LIN {X 0,Y 105.055,Z 539.774,A -85,B 0,C 180,E1 -26170.459,E2 -26170.459} C_VEL
LIN {X 0,Y 104.648,Z 537.475,A -85,B 0,C 180,E1 -26178.377,E2 -26178.377} C_VEL
LIN {X 0,Y 105.683,Z 533.747,A -85,B 0,C 180,E1 -26186.188,E2 -26186.188} C_VEL
LIN {X 0,Y 107.046,Z 529.972,A -85,B 0,C 180,E1 -26191.882,E2 -26191.882} C_VEL
LIN {X 0,Y 109.151,Z 525.302,A -85,B 0,C 180,E1 -26197.399,E2 -26197.399} C_VEL
LIN {X 0,Y 112.696,Z 518.5,A -85,B 0,C 180,E1 -26203.525,E2 -26203.525} C_VEL
LIN {X 0,Y 116.604,Z 511.397,A -85,B 0,C 180,E1 -26208.447,E2 -26208.447} C_VEL
LIN {X 0,Y 121.232,Z 502.855,A -85,B 0,C 180,E1 -26213.036,E2 -26213.036} C_VEL
LIN {X 0,Y 126.13,Z 493.405,A -85,B 0,C 180,E1 -26216.946,E2 -26216.946} C_VEL
LIN {X 0,Y 130.9,Z 483.256,A -85,B 0,C 180,E1 -26220.221,E2 -26220.221} C_VEL
LIN {X 0,Y 135.895,Z 470.856,A -85,B 0,C 180,E1 -26223.331,E2 -26223.331} C_VEL
LIN {X 0,Y 139.577,Z 460.327,A -85,B 0,C 180,E1 -26225.383,E2 -26225.383} C_VEL
LIN {X 0,Y 143.441,Z 448.136,A -85,B 0,C 180,E1 -26227.103,E2 -26227.103} C_VEL
LIN {X 0,Y 146.585,Z 434.369,A -85,B 0,C 180,E1 -26228.641,E2 -26228.641} C_VEL
LIN {X 0,Y 148.972,Z 420.343,A -85,B 0,C 180,E1 -26229.683,E2 -26229.683} C_VEL
LIN {X 0,Y 150.699,Z 403.652,A -85,B 0,C 180,E1 -26230.423,E2 -26230.423} C_VEL
LIN {X 0,Y 154.161,Z 361.132,A -85,B 0,C 180,E1 -26231.967,E2 -26231.967} C_VEL
LIN {X 0,Y 149.223,Z 350.379,A -85,B 0,C 180,E1 -26235.125,E2 -26235.125} C_VEL
LIN {X 0,Y 143.968,Z 340.636,A -85,B 0,C 180,E1 -26238.855,E2 -26238.855} C_VEL
LIN {X 0,Y 139.833,Z 333.875,A -85,B 0,C 180,E1 -26242.202,E2 -26242.202} C_VEL
LIN {X 0,Y 137.16,Z 329.846,A -85,B 0,C 180,E1 -26244.64,E2 -26244.64} C_VEL
LIN {X 0,Y 135.135,Z 326.776,A -85,B 0,C 180,E1 -26246.702,E2 -26246.702} C_VEL
LIN {X 0,Y 132.21,Z 322.641,A -85,B 0,C 180,E1 -26250.064,E2 -26250.064} C_VEL
LIN {X 0,Y 129.671,Z 319.416,A -85,B 0,C 180,E1 -26253.506,E2 -26253.506} C_VEL
LIN {X 0,Y 128.977,Z 318.09,A -85,B 0,C 180,E1 -26254.659,E2 -26254.659} C_VEL
LIN {X 0,Y 126.508,Z 315.752,A -85,B 0,C 180,E1 -26259.081,E2 -26259.081} C_VEL
LIN {X 0,Y 125.34,Z 312.869,A -85,B 0,C 180,E1 -26262.402,E2 -26262.402} C_VEL
LIN {X 0,Y 123.472,Z 311.706,A -85,B 0,C 180,E1 -26273.468,E2 -26273.468} C_VEL
LIN {X 0,Y 124.564,Z 312.157,A -85,B 0,C 180,E1 -26280.716,E2 -26280.716} C_VEL
LIN {X 0,Y 125.644,Z 313.032,A -85,B 0,C 180,E1 -26284.014,E2 -26284.014} C_VEL
LIN {X 0,Y 127.576,Z 316.671,A -85,B 0,C 180,E1 -26288.599,E2 -26288.599} C_VEL
LIN {X 0,Y 129.318,Z 318.362,A -85,B 0,C 180,E1 -26291.474,E2 -26291.474} C_VEL
LIN {X 0,Y 131.665,Z 322.03,A -85,B 0,C 180,E1 -26294.889,E2 -26294.889} C_VEL
LIN {X 0,Y 132.836,Z 323.455,A -85,B 0,C 180,E1 -26296.328,E2 -26296.328} C_VEL
LIN {X 0,Y 136.355,Z 328.602,A -85,B 0,C 180,E1 -26300.191,E2 -26300.191} C_VEL
LIN {X 0,Y 139.525,Z 333.327,A -85,B 0,C 180,E1 -26303.148,E2 -26303.148} C_VEL
LIN {X 0,Y 144.459,Z 341.575,A -85,B 0,C 180,E1 -26307.146,E2 -26307.146} C_VEL
LIN {X 0,Y 147.72,Z 347.787,A -85,B 0,C 180,E1 -26309.508,E2 -26309.508} C_VEL
LIN {X 0,Y 152.037,Z 359.604,A -85,B 0,C 180,E1 -26312.582,E2 -26312.582} C_VEL
LIN {X 0,Y 153.923,Z 365.668,A -85,B 0,C 180,E1 -26313.879,E2 -26313.879} C_VEL
LIN {X 0,Y 149.419,Z 421.282,A -85,B 0,C 180,E1 -26316.014,E2 -26316.014} C_VEL
LIN {X 0,Y 147.033,Z 436.247,A -85,B 0,C 180,E1 -26316.953,E2 -26316.953} C_VEL
LIN {X 0,Y 144.373,Z 447.938,A -85,B 0,C 180,E1 -26318.002,E2 -26318.002} C_VEL
LIN {X 0,Y 140.529,Z 461.489,A -85,B 0,C 180,E1 -26319.744,E2 -26319.744} C_VEL
LIN {X 0,Y 136.243,Z 473.608,A -85,B 0,C 180,E1 -26321.808,E2 -26321.808} C_VEL
LIN {X 0,Y 131.776,Z 485.158,A -85,B 0,C 180,E1 -26324.504,E2 -26324.504} C_VEL
LIN {X 0,Y 127.567,Z 494.106,A -85,B 0,C 180,E1 -26327.018,E2 -26327.018} C_VEL
LIN {X 0,Y 122.362,Z 504.452,A -85,B 0,C 180,E1 -26330.818,E2 -26330.818} C_VEL
LIN {X 0,Y 117.437,Z 513.807,A -85,B 0,C 180,E1 -26335.353,E2 -26335.353} C_VEL
LIN {X 0,Y 113.067,Z 521.924,A -85,B 0,C 180,E1 -26340.491,E2 -26340.491} C_VEL
LIN {X 0,Y 109.983,Z 528.046,A -85,B 0,C 180,E1 -26345.458,E2 -26345.458} C_VEL
LIN {X 0,Y 107.481,Z 533.33,A -85,B 0,C 180,E1 -26350.917,E2 -26350.917} C_VEL
LIN {X 0,Y 105.951,Z 537.632,A -85,B 0,C 180,E1 -26356.575,E2 -26356.575} C_VEL
LIN {X 0,Y 105.213,Z 541.041,A -85,B 0,C 180,E1 -26362.322,E2 -26362.322} C_VEL
LIN {X 0,Y 105.226,Z 544.198,A -85,B 0,C 180,E1 -26370,E2 -26370} C_VEL
LIN {X 0,Y 105.107,Z 545.222,A -85,B 0,C 180,E1 -26373.833,E2 -26373.833} C_VEL
LIN {X 0,Y 105.686,Z 546.264,A -85,B 0,C 180,E1 -26381.507,E2 -26381.507} C_VEL
LIN {X 0,Y 107.772,Z 546.007,A -85,B 0,C 180,E1 -26389.029,E2 -26389.029} C_VEL
LIN {X 0,Y 111.648,Z 544.464,A -85,B 0,C 180,E1 -26396.143,E2 -26396.143} C_VEL
LIN {X 0,Y 117.254,Z 541.466,A -85,B 0,C 180,E1 -26402.944,E2 -26402.944} C_VEL
LIN {X 0,Y 122.733,Z 538.083,A -85,B 0,C 180,E1 -26407.779,E2 -26407.779} C_VEL
LIN {X 0,Y 125.139,Z 536.162,A -85,B 0,C 180,E1 -26410.108,E2 -26410.108} C_VEL
LIN {X 0,Y 127.914,Z 532.718,A -85,B 0,C 180,E1 -26414.149,E2 -26414.149} C_VEL
LIN {X 0,Y 131.209,Z 528.811,A -85,B 0,C 180,E1 -26417.901,E2 -26417.901} C_VEL
LIN {X 0,Y 134.288,Z 526.052,A -85,B 0,C 180,E1 -26419.712,E2 -26419.712} C_VEL
LIN {X 0,Y 142.813,Z 518.685,A -85,B 0,C 180,E1 -26423.097,E2 -26423.097} C_VEL
LIN {X 0,Y 152.062,Z 509.256,A -85,B 0,C 180,E1 -26426.294,E2 -26426.294} C_VEL
LIN {X 0,Y 158.977,Z 501.172,A -85,B 0,C 180,E1 -26428.318,E2 -26428.318} C_VEL
LIN {X 0,Y 166.918,Z 490.585,A -85,B 0,C 180,E1 -26430.271,E2 -26430.271} C_VEL
LIN {X 0,Y 174.225,Z 478.929,A -85,B 0,C 180,E1 -26431.931,E2 -26431.931} C_VEL
LIN {X 0,Y 180.261,Z 467.528,A -85,B 0,C 180,E1 -26433.103,E2 -26433.103} C_VEL
LIN {X 0,Y 185.569,Z 455.21,A -85,B 0,C 180,E1 -26434.086,E2 -26434.086} C_VEL
LIN {X 0,Y 189.847,Z 442.69,A -85,B 0,C 180,E1 -26434.817,E2 -26434.817} C_VEL
LIN {X 0,Y 193.446,Z 428.393,A -85,B 0,C 180,E1 -26435.413,E2 -26435.413} C_VEL
LIN {X 0,Y 195.769,Z 413.722,A -85,B 0,C 180,E1 -26435.832,E2 -26435.832} C_VEL
LIN {X 0,Y 196.762,Z 403.98,A -85,B 0,C 180,E1 -26436.095,E2 -26436.095} C_VEL
LIN {X 0,Y 194.512,Z 396.884,A -85,B 0,C 180,E1 -26439.321,E2 -26439.321} C_VEL
LIN {X 0,Y 192.732,Z 391.862,A -85,B 0,C 180,E1 -26442.537,E2 -26442.537} C_VEL
LIN {X 0,Y 192.084,Z 390.368,A -85,B 0,C 180,E1 -26443.929,E2 -26443.929} C_VEL
LIN {X 0,Y 190.654,Z 386.905,A -85,B 0,C 180,E1 -26448.3,E2 -26448.3} C_VEL
LIN {X 0,Y 190.006,Z 386.116,A -85,B 0,C 180,E1 -26453.626,E2 -26453.626} C_VEL
LIN {X 0,Y 190.784,Z 386.681,A -85,B 0,C 180,E1 -26458.463,E2 -26458.463} C_VEL
LIN {X 0,Y 192.443,Z 390.776,A -85,B 0,C 180,E1 -26463.203,E2 -26463.203} C_VEL
LIN {X 0,Y 194.198,Z 394.785,A -85,B 0,C 180,E1 -26466.421,E2 -26466.421} C_VEL
LIN {X 0,Y 196.692,Z 400.396,A -85,B 0,C 180,E1 -26469.834,E2 -26469.834} C_VEL
LIN {X 0,Y 197,Z 401.105,A -85,B 0,C 180,E1 -26470.207,E2 -26470.207} C_VEL
LIN {X 0,Y 194.942,Z 418.493,A -85,B 0,C 180,E1 -26470.687,E2 -26470.687} C_VEL
LIN {X 0,Y 192.039,Z 432.581,A -85,B 0,C 180,E1 -26471.22,E2 -26471.22} C_VEL
LIN {X 0,Y 187.985,Z 446.274,A -85,B 0,C 180,E1 -26471.97,E2 -26471.97} C_VEL
LIN {X 0,Y 183.008,Z 459.186,A -85,B 0,C 180,E1 -26472.982,E2 -26472.982} C_VEL
LIN {X 0,Y 177.404,Z 470.841,A -85,B 0,C 180,E1 -26474.182,E2 -26474.182} C_VEL
LIN {X 0,Y 170.672,Z 482.429,A -85,B 0,C 180,E1 -26475.737,E2 -26475.737} C_VEL
LIN {X 0,Y 162.454,Z 494.275,A -85,B 0,C 180,E1 -26477.875,E2 -26477.875} C_VEL
LIN {X 0,Y 155.149,Z 503.119,A -85,B 0,C 180,E1 -26479.963,E2 -26479.963} C_VEL
LIN {X 0,Y 147.053,Z 511.638,A -85,B 0,C 180,E1 -26482.617,E2 -26482.617} C_VEL
LIN {X 0,Y 138.654,Z 519.319,A -85,B 0,C 180,E1 -26485.885,E2 -26485.885} C_VEL
LIN {X 0,Y 129.874,Z 526.245,A -85,B 0,C 180,E1 -26490.026,E2 -26490.026} C_VEL
LIN {X 0,Y 122.973,Z 530.956,A -85,B 0,C 180,E1 -26494.039,E2 -26494.039} C_VEL
LIN {X 0,Y 116.733,Z 534.675,A -85,B 0,C 180,E1 -26498.496,E2 -26498.496} C_VEL
LIN {X 0,Y 109.621,Z 538.24,A -85,B 0,C 180,E1 -26505.154,E2 -26505.154} C_VEL
LIN {X 0,Y 104.048,Z 540.303,A -85,B 0,C 180,E1 -26512.563,E2 -26512.563} C_VEL
LIN {X 0,Y 100.166,Z 540.919,A -85,B 0,C 180,E1 -26520.586,E2 -26520.586} C_VEL
LIN {X 0,Y 98.12,Z 540.097,A -85,B 0,C 180,E1 -26529.015,E2 -26529.015} C_VEL
LIN {X 0,Y 97.645,Z 539.166,A -85,B 0,C 180,E1 -26533.269,E2 -26533.269} C_VEL
LIN {X 0,Y 97.801,Z 536.251,A -85,B 0,C 180,E1 -26541.737,E2 -26541.737} C_VEL
LIN {X 0,Y 98.952,Z 532.993,A -85,B 0,C 180,E1 -26548.208,E2 -26548.208} C_VEL
LIN {X 0,Y 101.292,Z 527.59,A -85,B 0,C 180,E1 -26555.974,E2 -26555.974} C_VEL
LIN {X 0,Y 104.589,Z 521.332,A -85,B 0,C 180,E1 -26562.615,E2 -26562.615} C_VEL
LIN {X 0,Y 109.112,Z 513.53,A -85,B 0,C 180,E1 -26568.787,E2 -26568.787} C_VEL
LIN {X 0,Y 113.87,Z 505.378,A -85,B 0,C 180,E1 -26573.652,E2 -26573.652} C_VEL
LIN {X 0,Y 119.328,Z 495.55,A -85,B 0,C 180,E1 -26578.11,E2 -26578.11} C_VEL
LIN {X 0,Y 124.289,Z 485.719,A -85,B 0,C 180,E1 -26581.537,E2 -26581.537} C_VEL
LIN {X 0,Y 129.531,Z 473.872,A -85,B 0,C 180,E1 -26584.729,E2 -26584.729} C_VEL
LIN {X 0,Y 133.264,Z 463.878,A -85,B 0,C 180,E1 -26586.861,E2 -26586.861} C_VEL
LIN {X 0,Y 137.612,Z 451.509,A -85,B 0,C 180,E1 -26588.727,E2 -26588.727} C_VEL
LIN {X 0,Y 141.054,Z 438.037,A -85,B 0,C 180,E1 -26590.37,E2 -26590.37} C_VEL
LIN {X 0,Y 143.774,Z 423.832,A -85,B 0,C 180,E1 -26591.562,E2 -26591.562} C_VEL
LIN {X 0,Y 145.536,Z 409.73,A -85,B 0,C 180,E1 -26592.297,E2 -26592.297} C_VEL
LIN {X 0,Y 149.48,Z 363.624,A -85,B 0,C 180,E1 -26593.959,E2 -26593.959} C_VEL
LIN {X 0,Y 144.724,Z 353.294,A -85,B 0,C 180,E1 -26597.296,E2 -26597.296} C_VEL
LIN {X 0,Y 140.415,Z 345.116,A -85,B 0,C 180,E1 -26600.683,E2 -26600.683} C_VEL
LIN {X 0,Y 137.038,Z 339.424,A -85,B 0,C 180,E1 -26603.676,E2 -26603.676} C_VEL
LIN {X 0,Y 133.378,Z 333.414,A -85,B 0,C 180,E1 -26607.465,E2 -26607.465} C_VEL
LIN {X 0,Y 130.309,Z 329.05,A -85,B 0,C 180,E1 -26611.203,E2 -26611.203} C_VEL
LIN {X 0,Y 127.889,Z 325.615,A -85,B 0,C 180,E1 -26614.803,E2 -26614.803} C_VEL
LIN {X 0,Y 127.309,Z 324.749,A -85,B 0,C 180,E1 -26615.807,E2 -26615.807} C_VEL
LIN {X 0,Y 124.956,Z 322,A -85,B 0,C 180,E1 -26620.591,E2 -26620.591} C_VEL
LIN {X 0,Y 124.152,Z 319.832,A -85,B 0,C 180,E1 -26623.212,E2 -26623.212} C_VEL
LIN {X 0,Y 122.594,Z 318.744,A -85,B 0,C 180,E1 -26633.421,E2 -26633.421} C_VEL
LIN {X 0,Y 123.676,Z 319.227,A -85,B 0,C 180,E1 -26640.721,E2 -26640.721} C_VEL
LIN {X 0,Y 124.458,Z 319.88,A -85,B 0,C 180,E1 -26643.241,E2 -26643.241} C_VEL
LIN {X 0,Y 126.27,Z 323.471,A -85,B 0,C 180,E1 -26647.892,E2 -26647.892} C_VEL
LIN {X 0,Y 127.746,Z 325.017,A -85,B 0,C 180,E1 -26650.506,E2 -26650.506} C_VEL
LIN {X 0,Y 129.988,Z 328.613,A -85,B 0,C 180,E1 -26653.986,E2 -26653.986} C_VEL
LIN {X 0,Y 131.059,Z 330.091,A -85,B 0,C 180,E1 -26655.407,E2 -26655.407} C_VEL
LIN {X 0,Y 134.171,Z 334.838,A -85,B 0,C 180,E1 -26659.064,E2 -26659.064} C_VEL
LIN {X 0,Y 137.629,Z 340.206,A -85,B 0,C 180,E1 -26662.482,E2 -26662.482} C_VEL
LIN {X 0,Y 142.336,Z 348.768,A -85,B 0,C 180,E1 -26666.513,E2 -26666.513} C_VEL
LIN {X 0,Y 144.393,Z 353.04,A -85,B 0,C 180,E1 -26668.115,E2 -26668.115} C_VEL
LIN {X 0,Y 148.226,Z 364.194,A -85,B 0,C 180,E1 -26671.091,E2 -26671.091} C_VEL
LIN {X 0,Y 149.316,Z 367.945,A -85,B 0,C 180,E1 -26671.922,E2 -26671.922} C_VEL
LIN {X 0,Y 144.667,Z 421.831,A -85,B 0,C 180,E1 -26673.975,E2 -26673.975} C_VEL
LIN {X 0,Y 142.198,Z 436.497,A -85,B 0,C 180,E1 -26674.904,E2 -26674.904} C_VEL
LIN {X 0,Y 139.441,Z 448.072,A -85,B 0,C 180,E1 -26675.947,E2 -26675.947} C_VEL
LIN {X 0,Y 135.446,Z 461.552,A -85,B 0,C 180,E1 -26677.695,E2 -26677.695} C_VEL
LIN {X 0,Y 130.648,Z 474.492,A -85,B 0,C 180,E1 -26679.956,E2 -26679.956} C_VEL
LIN {X 0,Y 125.636,Z 486.47,A -85,B 0,C 180,E1 -26682.847,E2 -26682.847} C_VEL
LIN {X 0,Y 121.889,Z 494.056,A -85,B 0,C 180,E1 -26685.064,E2 -26685.064} C_VEL
LIN {X 0,Y 116.896,Z 503.526,A -85,B 0,C 180,E1 -26688.599,E2 -26688.599} C_VEL
LIN {X 0,Y 111.6,Z 513.018,A -85,B 0,C 180,E1 -26693.255,E2 -26693.255} C_VEL
LIN {X 0,Y 106.607,Z 521.741,A -85,B 0,C 180,E1 -26698.991,E2 -26698.991} C_VEL
LIN {X 0,Y 102.51,Z 529.312,A -85,B 0,C 180,E1 -26705.71,E2 -26705.71} C_VEL
LIN {X 0,Y 100.048,Z 534.366,A -85,B 0,C 180,E1 -26711.572,E2 -26711.572} C_VEL
LIN {X 0,Y 98.66,Z 538.424,A -85,B 0,C 180,E1 -26717.66,E2 -26717.66} C_VEL
LIN {X 0,Y 98.168,Z 540.628,A -85,B 0,C 180,E1 -26721.768,E2 -26721.768} C_VEL
LIN {X 0,Y 98.144,Z 543.879,A -85,B 0,C 180,E1 -26730,E2 -26730} C_VEL
LIN {X 0,Y 98.016,Z 544.936,A -85,B 0,C 180,E1 -26734.111,E2 -26734.111} C_VEL
LIN {X 0,Y 98.71,Z 546.046,A -85,B 0,C 180,E1 -26742.332,E2 -26742.332} C_VEL
LIN {X 0,Y 101.044,Z 545.858,A -85,B 0,C 180,E1 -26750.35,E2 -26750.35} C_VEL
LIN {X 0,Y 105.277,Z 544.386,A -85,B 0,C 180,E1 -26757.858,E2 -26757.858} C_VEL
LIN {X 0,Y 111.095,Z 541.599,A -85,B 0,C 180,E1 -26764.704,E2 -26764.704} C_VEL
LIN {X 0,Y 118.371,Z 537.421,A -85,B 0,C 180,E1 -26770.774,E2 -26770.774} C_VEL
LIN {X 0,Y 126.87,Z 531.729,A -85,B 0,C 180,E1 -26776.064,E2 -26776.064} C_VEL
LIN {X 0,Y 134.288,Z 526.052,A -85,B 0,C 180,E1 -26779.712,E2 -26779.712} C_VEL
LIN {X 0,Y 137.468,Z 523.137,A -85,B 0,C 180,E1 -26781.406,E2 -26781.406} C_VEL
LIN {X 0,Y 141.503,Z 518.157,A -85,B 0,C 180,E1 -26784.522,E2 -26784.522} C_VEL
LIN {X 0,Y 145.626,Z 512.784,A -85,B 0,C 180,E1 -26787.415,E2 -26787.415} C_VEL
LIN {X 0,Y 148.825,Z 509.125,A -85,B 0,C 180,E1 -26788.739,E2 -26788.739} C_VEL
LIN {X 0,Y 156.857,Z 500.005,A -85,B 0,C 180,E1 -26790.889,E2 -26790.889} C_VEL
LIN {X 0,Y 165.016,Z 489.23,A -85,B 0,C 180,E1 -26792.753,E2 -26792.753} C_VEL
LIN {X 0,Y 172.546,Z 477.332,A -85,B 0,C 180,E1 -26794.31,E2 -26794.31} C_VEL
LIN {X 0,Y 178.753,Z 465.609,A -85,B 0,C 180,E1 -26795.392,E2 -26795.392} C_VEL
LIN {X 0,Y 184.17,Z 452.859,A -85,B 0,C 180,E1 -26796.323,E2 -26796.323} C_VEL
LIN {X 0,Y 188.709,Z 439.079,A -85,B 0,C 180,E1 -26797.028,E2 -26797.028} C_VEL
LIN {X 0,Y 192.069,Z 424.637,A -85,B 0,C 180,E1 -26797.529,E2 -26797.529} C_VEL
LIN {X 0,Y 194.267,Z 408.43,A -85,B 0,C 180,E1 -26797.963,E2 -26797.963} C_VEL
LIN {X 0,Y 194.236,Z 407.484,A -85,B 0,C 180,E1 -26798.123,E2 -26798.123} C_VEL
LIN {X 0,Y 192.575,Z 401.945,A -85,B 0,C 180,E1 -26800.915,E2 -26800.915} C_VEL
LIN {X 0,Y 191.205,Z 397.652,A -85,B 0,C 180,E1 -26803.853,E2 -26803.853} C_VEL
LIN {X 0,Y 189.649,Z 393.858,A -85,B 0,C 180,E1 -26808.779,E2 -26808.779} C_VEL
LIN {X 0,Y 189.128,Z 393.156,A -85,B 0,C 180,E1 -26813.597,E2 -26813.597} C_VEL
LIN {X 0,Y 189.814,Z 393.751,A -85,B 0,C 180,E1 -26818.189,E2 -26818.189} C_VEL
LIN {X 0,Y 191.248,Z 397.539,A -85,B 0,C 180,E1 -26822.622,E2 -26822.622} C_VEL
LIN {X 0,Y 192.906,Z 401.537,A -85,B 0,C 180,E1 -26825.878,E2 -26825.878} C_VEL
LIN {X 0,Y 194.531,Z 405.466,A -85,B 0,C 180,E1 -26828.342,E2 -26828.342} C_VEL
LIN {X 0,Y 192.325,Z 421.692,A -85,B 0,C 180,E1 -26828.778,E2 -26828.778} C_VEL
LIN {X 0,Y 189.209,Z 435.402,A -85,B 0,C 180,E1 -26829.318,E2 -26829.318} C_VEL
LIN {X 0,Y 185.111,Z 448.303,A -85,B 0,C 180,E1 -26830.027,E2 -26830.027} C_VEL
LIN {X 0,Y 179.889,Z 461.11,A -85,B 0,C 180,E1 -26831.017,E2 -26831.017} C_VEL
LIN {X 0,Y 173.38,Z 473.823,A -85,B 0,C 180,E1 -26832.338,E2 -26832.338} C_VEL
LIN {X 0,Y 166.483,Z 484.922,A -85,B 0,C 180,E1 -26833.855,E2 -26833.855} C_VEL
LIN {X 0,Y 158.806,Z 495.348,A -85,B 0,C 180,E1 -26835.735,E2 -26835.735} C_VEL
LIN {X 0,Y 149.8,Z 505.625,A -85,B 0,C 180,E1 -26838.192,E2 -26838.192} C_VEL
LIN {X 0,Y 141.136,Z 514.091,A -85,B 0,C 180,E1 -26840.99,E2 -26840.99} C_VEL
LIN {X 0,Y 131.521,Z 522.122,A -85,B 0,C 180,E1 -26844.716,E2 -26844.716} C_VEL
LIN {X 0,Y 123.771,Z 527.666,A -85,B 0,C 180,E1 -26848.346,E2 -26848.346} C_VEL
LIN {X 0,Y 115.504,Z 532.787,A -85,B 0,C 180,E1 -26853.198,E2 -26853.198} C_VEL
LIN {X 0,Y 108.144,Z 536.612,A -85,B 0,C 180,E1 -26858.756,E2 -26858.756} C_VEL
LIN {X 0,Y 101.094,Z 539.507,A -85,B 0,C 180,E1 -26865.959,E2 -26865.959} C_VEL
LIN {X 0,Y 95.773,Z 540.937,A -85,B 0,C 180,E1 -26874.053,E2 -26874.053} C_VEL
LIN {X 0,Y 92.25,Z 540.947,A -85,B 0,C 180,E1 -26882.801,E2 -26882.801} C_VEL
LIN {X 0,Y 91.233,Z 540.377,A -85,B 0,C 180,E1 -26887.561,E2 -26887.561} C_VEL
LIN {X 0,Y 90.395,Z 538.294,A -85,B 0,C 180,E1 -26896.513,E2 -26896.513} C_VEL
LIN {X 0,Y 90.633,Z 536.702,A -85,B 0,C 180,E1 -26901.079,E2 -26901.079} C_VEL
LIN {X 0,Y 91.502,Z 534.187,A -85,B 0,C 180,E1 -26906.729,E2 -26906.729} C_VEL
LIN {X 0,Y 93.419,Z 529.722,A -85,B 0,C 180,E1 -26914.315,E2 -26914.315} C_VEL
LIN {X 0,Y 95.995,Z 524.88,A -85,B 0,C 180,E1 -26920.547,E2 -26920.547} C_VEL
LIN {X 0,Y 100.237,Z 517.884,A -85,B 0,C 180,E1 -26927.337,E2 -26927.337} C_VEL
LIN {X 0,Y 105.651,Z 509.214,A -85,B 0,C 180,E1 -26933.523,E2 -26933.523} C_VEL
LIN {X 0,Y 111.121,Z 500.145,A -85,B 0,C 180,E1 -26938.317,E2 -26938.317} C_VEL
LIN {X 0,Y 116.512,Z 490.446,A -85,B 0,C 180,E1 -26942.212,E2 -26942.212} C_VEL
LIN {X 0,Y 121.556,Z 480.373,A -85,B 0,C 180,E1 -26945.322,E2 -26945.322} C_VEL
LIN {X 0,Y 125.966,Z 470.098,A -85,B 0,C 180,E1 -26947.859,E2 -26947.859} C_VEL
LIN {X 0,Y 130.098,Z 459.279,A -85,B 0,C 180,E1 -26949.903,E2 -26949.903} C_VEL
LIN {X 0,Y 133.948,Z 447.832,A -85,B 0,C 180,E1 -26951.483,E2 -26951.483} C_VEL
LIN {X 0,Y 137.361,Z 433.914,A -85,B 0,C 180,E1 -26953.003,E2 -26953.003} C_VEL
LIN {X 0,Y 139.944,Z 419.476,A -85,B 0,C 180,E1 -26954.035,E2 -26954.035} C_VEL
LIN {X 0,Y 141.963,Z 400.009,A -85,B 0,C 180,E1 -26954.858,E2 -26954.858} C_VEL
LIN {X 0,Y 144.953,Z 366.379,A -85,B 0,C 180,E1 -26956.06,E2 -26956.06} C_VEL
LIN {X 0,Y 140.951,Z 357.341,A -85,B 0,C 180,E1 -26959.176,E2 -26959.176} C_VEL
LIN {X 0,Y 136.566,Z 348.776,A -85,B 0,C 180,E1 -26963.023,E2 -26963.023} C_VEL
LIN {X 0,Y 132.612,Z 341.948,A -85,B 0,C 180,E1 -26967.089,E2 -26967.089} C_VEL
LIN {X 0,Y 130.337,Z 338.348,A -85,B 0,C 180,E1 -26969.806,E2 -26969.806} C_VEL
LIN {X 0,Y 128.578,Z 335.578,A -85,B 0,C 180,E1 -26972.208,E2 -26972.208} C_VEL
LIN {X 0,Y 126.213,Z 331.959,A -85,B 0,C 180,E1 -26976.047,E2 -26976.047} C_VEL
LIN {X 0,Y 123.558,Z 328.361,A -85,B 0,C 180,E1 -26981.941,E2 -26981.941} C_VEL
LIN {X 0,Y 123.044,Z 326.809,A -85,B 0,C 180,E1 -26983.868,E2 -26983.868} C_VEL
LIN {X 0,Y 121.715,Z 325.794,A -85,B 0,C 180,E1 -26993.373,E2 -26993.373} C_VEL
LIN {X 0,Y 122.787,Z 326.295,A -85,B 0,C 180,E1 -27000.726,E2 -27000.726} C_VEL
LIN {X 0,Y 123.321,Z 326.891,A -85,B 0,C 180,E1 -27002.585,E2 -27002.585} C_VEL
LIN {X 0,Y 125.18,Z 330.497,A -85,B 0,C 180,E1 -27007.575,E2 -27007.575} C_VEL
LIN {X 0,Y 126.265,Z 331.771,A -85,B 0,C 180,E1 -27009.617,E2 -27009.617} C_VEL
LIN {X 0,Y 129.318,Z 336.717,A -85,B 0,C 180,E1 -27014.461,E2 -27014.461} C_VEL
LIN {X 0,Y 132.216,Z 341.351,A -85,B 0,C 180,E1 -27018.101,E2 -27018.101} C_VEL
LIN {X 0,Y 135.313,Z 346.514,A -85,B 0,C 180,E1 -27021.389,E2 -27021.389} C_VEL
LIN {X 0,Y 139.753,Z 354.991,A -85,B 0,C 180,E1 -27025.46,E2 -27025.46} C_VEL
LIN {X 0,Y 141.233,Z 358.587,A -85,B 0,C 180,E1 -27026.737,E2 -27026.737} C_VEL
LIN {X 0,Y 144.742,Z 369.668,A -85,B 0,C 180,E1 -27029.722,E2 -27029.722} C_VEL
LIN {X 0,Y 144.279,Z 376.579,A -85,B 0,C 180,E1 -27030.049,E2 -27030.049} C_VEL
LIN {X 0,Y 140.22,Z 421.254,A -85,B 0,C 180,E1 -27031.736,E2 -27031.736} C_VEL
LIN {X 0,Y 137.73,Z 435.872,A -85,B 0,C 180,E1 -27032.655,E2 -27032.655} C_VEL
LIN {X 0,Y 134.701,Z 448.125,A -85,B 0,C 180,E1 -27033.744,E2 -27033.744} C_VEL
LIN {X 0,Y 130.551,Z 461.558,A -85,B 0,C 180,E1 -27035.49,E2 -27035.49} C_VEL
LIN {X 0,Y 125.55,Z 474.462,A -85,B 0,C 180,E1 -27037.752,E2 -27037.752} C_VEL
LIN {X 0,Y 120.391,Z 486.245,A -85,B 0,C 180,E1 -27040.634,E2 -27040.634} C_VEL
LIN {X 0,Y 116.361,Z 493.981,A -85,B 0,C 180,E1 -27042.919,E2 -27042.919} C_VEL
LIN {X 0,Y 110.605,Z 504.282,A -85,B 0,C 180,E1 -27046.917,E2 -27046.917} C_VEL
LIN {X 0,Y 105.071,Z 513.603,A -85,B 0,C 180,E1 -27051.778,E2 -27051.778} C_VEL
LIN {X 0,Y 100.098,Z 521.709,A -85,B 0,C 180,E1 -27057.417,E2 -27057.417} C_VEL
LIN {X 0,Y 96.004,Z 528.717,A -85,B 0,C 180,E1 -27063.945,E2 -27063.945} C_VEL
LIN {X 0,Y 93.285,Z 533.856,A -85,B 0,C 180,E1 -27070.183,E2 -27070.183} C_VEL
LIN {X 0,Y 91.359,Z 539.125,A -85,B 0,C 180,E1 -27078.912,E2 -27078.912} C_VEL
LIN {X 0,Y 90.876,Z 542.054,A -85,B 0,C 180,E1 -27085.564,E2 -27085.564} C_VEL
LIN {X 0,Y 91.049,Z 543.542,A -85,B 0,C 180,E1 -27089.999,E2 -27089.999} C_VEL
LIN {X 0,Y 90.923,Z 544.64,A -85,B 0,C 180,E1 -27094.433,E2 -27094.433} C_VEL
LIN {X 0,Y 91.767,Z 545.825,A -85,B 0,C 180,E1 -27103.282,E2 -27103.282} C_VEL
LIN {X 0,Y 94.377,Z 545.71,A -85,B 0,C 180,E1 -27111.859,E2 -27111.859} C_VEL
LIN {X 0,Y 99.015,Z 544.313,A -85,B 0,C 180,E1 -27119.791,E2 -27119.791} C_VEL
LIN {X 0,Y 105.306,Z 541.601,A -85,B 0,C 180,E1 -27126.915,E2 -27126.915} C_VEL
LIN {X 0,Y 113.08,Z 537.502,A -85,B 0,C 180,E1 -27133.129,E2 -27133.129} C_VEL
LIN {X 0,Y 122.034,Z 531.895,A -85,B 0,C 180,E1 -27138.474,E2 -27138.474} C_VEL
LIN {X 0,Y 130.732,Z 525.607,A -85,B 0,C 180,E1 -27142.459,E2 -27142.459} C_VEL
LIN {X 0,Y 140.037,Z 517.816,A -85,B 0,C 180,E1 -27145.9,E2 -27145.9} C_VEL
LIN {X 0,Y 148.825,Z 509.125,A -85,B 0,C 180,E1 -27148.739,E2 -27148.739} C_VEL
LIN {X 0,Y 152.036,Z 505.343,A -85,B 0,C 180,E1 -27149.973,E2 -27149.973} C_VEL
LIN {X 0,Y 156.334,Z 499.018,A -85,B 0,C 180,E1 -27152.329,E2 -27152.329} C_VEL
LIN {X 0,Y 160.557,Z 492.241,A -85,B 0,C 180,E1 -27154.432,E2 -27154.432} C_VEL
LIN {X 0,Y 163.538,Z 487.763,A -85,B 0,C 180,E1 -27155.273,E2 -27155.273} C_VEL
LIN {X 0,Y 171.19,Z 475.674,A -85,B 0,C 180,E1 -27156.715,E2 -27156.715} C_VEL
LIN {X 0,Y 177.521,Z 463.606,A -85,B 0,C 180,E1 -27157.727,E2 -27157.727} C_VEL
LIN {X 0,Y 182.742,Z 451.206,A -85,B 0,C 180,E1 -27158.529,E2 -27158.529} C_VEL
LIN {X 0,Y 187.302,Z 437.036,A -85,B 0,C 180,E1 -27159.187,E2 -27159.187} C_VEL
LIN {X 0,Y 190.593,Z 422.367,A -85,B 0,C 180,E1 -27159.646,E2 -27159.646} C_VEL
LIN {X 0,Y 192.076,Z 411.714,A -85,B 0,C 180,E1 -27159.945,E2 -27159.945} C_VEL
LIN {X 0,Y 191.014,Z 407.835,A -85,B 0,C 180,E1 -27162.063,E2 -27162.063} C_VEL
LIN {X 0,Y 190.03,Z 404.356,A -85,B 0,C 180,E1 -27164.461,E2 -27164.461} C_VEL
LIN {X 0,Y 188.659,Z 400.795,A -85,B 0,C 180,E1 -27169.263,E2 -27169.263} C_VEL
LIN {X 0,Y 188.248,Z 400.206,A -85,B 0,C 180,E1 -27173.567,E2 -27173.567} C_VEL
LIN {X 0,Y 188.846,Z 400.735,A -85,B 0,C 180,E1 -27177.864,E2 -27177.864} C_VEL
LIN {X 0,Y 190.07,Z 404.232,A -85,B 0,C 180,E1 -27182.01,E2 -27182.01} C_VEL
LIN {X 0,Y 191.549,Z 408.123,A -85,B 0,C 180,E1 -27185.184,E2 -27185.184} C_VEL
LIN {X 0,Y 192.251,Z 410.002,A -85,B 0,C 180,E1 -27186.425,E2 -27186.425} C_VEL
LIN {X 0,Y 189.906,Z 424.706,A -85,B 0,C 180,E1 -27186.815,E2 -27186.815} C_VEL
LIN {X 0,Y 186.189,Z 439.241,A -85,B 0,C 180,E1 -27187.4,E2 -27187.4} C_VEL
LIN {X 0,Y 181.493,Z 452.609,A -85,B 0,C 180,E1 -27188.175,E2 -27188.175} C_VEL
LIN {X 0,Y 175.689,Z 465.48,A -85,B 0,C 180,E1 -27189.204,E2 -27189.204} C_VEL
LIN {X 0,Y 168.872,Z 477.696,A -85,B 0,C 180,E1 -27190.524,E2 -27190.524} C_VEL
LIN {X 0,Y 160.896,Z 489.486,A -85,B 0,C 180,E1 -27192.225,E2 -27192.225} C_VEL
LIN {X 0,Y 152.265,Z 500.044,A -85,B 0,C 180,E1 -27194.244,E2 -27194.244} C_VEL
LIN {X 0,Y 142.795,Z 509.794,A -85,B 0,C 180,E1 -27196.814,E2 -27196.814} C_VEL
LIN {X 0,Y 132.824,Z 518.494,A -85,B 0,C 180,E1 -27200.089,E2 -27200.089} C_VEL
LIN {X 0,Y 123.079,Z 525.671,A -85,B 0,C 180,E1 -27203.993,E2 -27203.993} C_VEL
LIN {X 0,Y 115.243,Z 530.579,A -85,B 0,C 180,E1 -27207.842,E2 -27207.842} C_VEL
LIN {X 0,Y 105.782,Z 535.588,A -85,B 0,C 180,E1 -27213.854,E2 -27213.854} C_VEL
LIN {X 0,Y 98.691,Z 538.576,A -85,B 0,C 180,E1 -27219.852,E2 -27219.852} C_VEL
LIN {X 0,Y 92.594,Z 540.5,A -85,B 0,C 180,E1 -27226.914,E2 -27226.914} C_VEL
LIN {X 0,Y 87.517,Z 541.306,A -85,B 0,C 180,E1 -27235.798,E2 -27235.798} C_VEL
LIN {X 0,Y 84.474,Z 540.702,A -85,B 0,C 180,E1 -27245.42,E2 -27245.42} C_VEL
LIN {X 0,Y 83.664,Z 539.877,A -85,B 0,C 180,E1 -27250.367,E2 -27250.367} C_VEL
LIN {X 0,Y 83.46,Z 537.148,A -85,B 0,C 180,E1 -27260.305,E2 -27260.305} C_VEL
LIN {X 0,Y 84.43,Z 534.358,A -85,B 0,C 180,E1 -27267.152,E2 -27267.152} C_VEL
LIN {X 0,Y 86.285,Z 530.302,A -85,B 0,C 180,E1 -27274.672,E2 -27274.672} C_VEL
LIN {X 0,Y 89,Z 525.561,A -85,B 0,C 180,E1 -27281.386,E2 -27281.386} C_VEL
LIN {X 0,Y 93.477,Z 518.675,A -85,B 0,C 180,E1 -27288.635,E2 -27288.635} C_VEL
LIN {X 0,Y 98.294,Z 511.492,A -85,B 0,C 180,E1 -27294.275,E2 -27294.275} C_VEL
LIN {X 0,Y 103.919,Z 502.841,A -85,B 0,C 180,E1 -27299.361,E2 -27299.361} C_VEL
LIN {X 0,Y 110.164,Z 492.435,A -85,B 0,C 180,E1 -27303.887,E2 -27303.887} C_VEL
LIN {X 0,Y 115.861,Z 481.809,A -85,B 0,C 180,E1 -27307.343,E2 -27307.343} C_VEL
LIN {X 0,Y 121.051,Z 470.379,A -85,B 0,C 180,E1 -27310.232,E2 -27310.232} C_VEL
LIN {X 0,Y 125.371,Z 459.579,A -85,B 0,C 180,E1 -27312.274,E2 -27312.274} C_VEL
LIN {X 0,Y 129.377,Z 448.156,A -85,B 0,C 180,E1 -27313.836,E2 -27313.836} C_VEL
LIN {X 0,Y 133.001,Z 433.964,A -85,B 0,C 180,E1 -27315.374,E2 -27315.374} C_VEL
LIN {X 0,Y 135.636,Z 419.834,A -85,B 0,C 180,E1 -27316.368,E2 -27316.368} C_VEL
LIN {X 0,Y 137.774,Z 399.911,A -85,B 0,C 180,E1 -27317.208,E2 -27317.208} C_VEL
LIN {X 0,Y 140.588,Z 368.945,A -85,B 0,C 180,E1 -27318.332,E2 -27318.332} C_VEL
LIN {X 0,Y 136.901,Z 360.508,A -85,B 0,C 180,E1 -27321.551,E2 -27321.551} C_VEL
LIN {X 0,Y 132.961,Z 352.576,A -85,B 0,C 180,E1 -27325.473,E2 -27325.473} C_VEL
LIN {X 0,Y 129.272,Z 345.907,A -85,B 0,C 180,E1 -27329.854,E2 -27329.854} C_VEL
LIN {X 0,Y 126.624,Z 341.738,A -85,B 0,C 180,E1 -27333.644,E2 -27333.644} C_VEL
LIN {X 0,Y 124.382,Z 338.17,A -85,B 0,C 180,E1 -27337.71,E2 -27337.71} C_VEL
LIN {X 0,Y 122.325,Z 335.006,A -85,B 0,C 180,E1 -27342.954,E2 -27342.954} C_VEL
LIN {X 0,Y 121.926,Z 333.745,A -85,B 0,C 180,E1 -27344.638,E2 -27344.638} C_VEL
LIN {X 0,Y 120.839,Z 332.818,A -85,B 0,C 180,E1 -27353.325,E2 -27353.325} C_VEL
LIN {X 0,Y 121.838,Z 333.284,A -85,B 0,C 180,E1 -27360.484,E2 -27360.484} C_VEL
LIN {X 0,Y 122.249,Z 333.975,A -85,B 0,C 180,E1 -27362.088,E2 -27362.088} C_VEL
LIN {X 0,Y 124.17,Z 337.615,A -85,B 0,C 180,E1 -27367.41,E2 -27367.41} C_VEL
LIN {X 0,Y 124.867,Z 338.61,A -85,B 0,C 180,E1 -27368.816,E2 -27368.816} C_VEL
LIN {X 0,Y 127.459,Z 343.002,A -85,B 0,C 180,E1 -27373.253,E2 -27373.253} C_VEL
LIN {X 0,Y 130.336,Z 347.927,A -85,B 0,C 180,E1 -27377.155,E2 -27377.155} C_VEL
LIN {X 0,Y 132.99,Z 352.72,A -85,B 0,C 180,E1 -27380.196,E2 -27380.196} C_VEL
LIN {X 0,Y 136.784,Z 360.322,A -85,B 0,C 180,E1 -27383.972,E2 -27383.972} C_VEL
LIN {X 0,Y 138.26,Z 364.518,A -85,B 0,C 180,E1 -27385.401,E2 -27385.401} C_VEL
LIN {X 0,Y 140.498,Z 372.041,A -85,B 0,C 180,E1 -27387.518,E2 -27387.518} C_VEL
LIN {X 0,Y 136.063,Z 420.3,A -85,B 0,C 180,E1 -27389.353,E2 -27389.353} C_VEL
LIN {X 0,Y 133.659,Z 434.429,A -85,B 0,C 180,E1 -27390.197,E2 -27390.197} C_VEL
LIN {X 0,Y 130.535,Z 447.01,A -85,B 0,C 180,E1 -27391.273,E2 -27391.273} C_VEL
LIN {X 0,Y 126.516,Z 459.737,A -85,B 0,C 180,E1 -27392.841,E2 -27392.841} C_VEL
LIN {X 0,Y 121.266,Z 472.945,A -85,B 0,C 180,E1 -27395.055,E2 -27395.055} C_VEL
LIN {X 0,Y 115.87,Z 484.974,A -85,B 0,C 180,E1 -27397.955,E2 -27397.955} C_VEL
LIN {X 0,Y 111.019,Z 493.876,A -85,B 0,C 180,E1 -27400.567,E2 -27400.567} C_VEL
LIN {X 0,Y 105.486,Z 503.325,A -85,B 0,C 180,E1 -27404.257,E2 -27404.257} C_VEL
LIN {X 0,Y 99.518,Z 512.778,A -85,B 0,C 180,E1 -27409.214,E2 -27409.214} C_VEL
LIN {X 0,Y 93.7,Z 521.624,A -85,B 0,C 180,E1 -27415.604,E2 -27415.604} C_VEL
LIN {X 0,Y 89.607,Z 528.1,A -85,B 0,C 180,E1 -27421.928,E2 -27421.928} C_VEL
LIN {X 0,Y 86.598,Z 533.303,A -85,B 0,C 180,E1 -27428.58,E2 -27428.58} C_VEL
LIN {X 0,Y 84.74,Z 537.473,A -85,B 0,C 180,E1 -27435.593,E2 -27435.593} C_VEL
LIN {X 0,Y 84.104,Z 539.76,A -85,B 0,C 180,E1 -27440.379,E2 -27440.379} C_VEL
LIN {X 0,Y 83.947,Z 543.178,A -85,B 0,C 180,E1 -27449.999,E2 -27449.999} C_VEL
LIN {X 0,Y 83.854,Z 544.317,A -85,B 0,C 180,E1 -27454.807,E2 -27454.807} C_VEL
LIN {X 0,Y 84.832,Z 545.58,A -85,B 0,C 180,E1 -27464.39,E2 -27464.39} C_VEL
LIN {X 0,Y 87.789,Z 545.544,A -85,B 0,C 180,E1 -27473.594,E2 -27473.594} C_VEL
LIN {X 0,Y 92.885,Z 544.228,A -85,B 0,C 180,E1 -27481.98,E2 -27481.98} C_VEL
LIN {X 0,Y 99.696,Z 541.602,A -85,B 0,C 180,E1 -27489.378,E2 -27489.378} C_VEL
LIN {X 0,Y 107.978,Z 537.584,A -85,B 0,C 180,E1 -27495.72,E2 -27495.72} C_VEL
LIN {X 0,Y 117.431,Z 532.06,A -85,B 0,C 180,E1 -27501.077,E2 -27501.077} C_VEL
LIN {X 0,Y 126.538,Z 525.863,A -85,B 0,C 180,E1 -27505.005,E2 -27505.005} C_VEL
LIN {X 0,Y 136.186,Z 518.174,A -85,B 0,C 180,E1 -27508.372,E2 -27508.372} C_VEL
LIN {X 0,Y 146.131,Z 508.725,A -85,B 0,C 180,E1 -27511.365,E2 -27511.365} C_VEL
LIN {X 0,Y 153.547,Z 500.608,A -85,B 0,C 180,E1 -27513.19,E2 -27513.19} C_VEL
LIN {X 0,Y 161.911,Z 489.993,A -85,B 0,C 180,E1 -27514.97,E2 -27514.97} C_VEL
LIN {X 0,Y 163.538,Z 487.763,A -85,B 0,C 180,E1 -27515.273,E2 -27515.273} C_VEL
LIN {X 0,Y 165.392,Z 484.702,A -85,B 0,C 180,E1 -27515.893,E2 -27515.893} C_VEL
LIN {X 0,Y 167.51,Z 479.998,A -85,B 0,C 180,E1 -27517.409,E2 -27517.409} C_VEL
LIN {X 0,Y 169.589,Z 475.207,A -85,B 0,C 180,E1 -27518.848,E2 -27518.848} C_VEL
LIN {X 0,Y 171.297,Z 471.893,A -85,B 0,C 180,E1 -27519.347,E2 -27519.347} C_VEL
LIN {X 0,Y 177.382,Z 459.801,A -85,B 0,C 180,E1 -27520.214,E2 -27520.214} C_VEL
LIN {X 0,Y 183.046,Z 445.51,A -85,B 0,C 180,E1 -27520.97,E2 -27520.97} C_VEL
LIN {X 0,Y 187.095,Z 431.514,A -85,B 0,C 180,E1 -27521.493,E2 -27521.493} C_VEL
LIN {X 0,Y 189.89,Z 416.933,A -85,B 0,C 180,E1 -27521.868,E2 -27521.868} C_VEL
LIN {X 0,Y 189.999,Z 415.756,A -85,B 0,C 180,E1 -27521.969,E2 -27521.969} C_VEL
LIN {X 0,Y 188.933,Z 411.275,A -85,B 0,C 180,E1 -27524.904,E2 -27524.904} C_VEL
LIN {X 0,Y 187.788,Z 407.867,A -85,B 0,C 180,E1 -27529.212,E2 -27529.212} C_VEL
LIN {X 0,Y 187.369,Z 407.247,A -85,B 0,C 180,E1 -27533.536,E2 -27533.536} C_VEL
LIN {X 0,Y 187.892,Z 407.764,A -85,B 0,C 180,E1 -27537.585,E2 -27537.585} C_VEL
LIN {X 0,Y 188.904,Z 410.949,A -85,B 0,C 180,E1 -27541.384,E2 -27541.384} C_VEL
LIN {X 0,Y 190.094,Z 414.543,A -85,B 0,C 180,E1 -27544.4,E2 -27544.4} C_VEL
LIN {X 0,Y 187.36,Z 429.181,A -85,B 0,C 180,E1 -27544.863,E2 -27544.863} C_VEL
LIN {X 0,Y 183.539,Z 442.576,A -85,B 0,C 180,E1 -27545.404,E2 -27545.404} C_VEL
LIN {X 0,Y 178.494,Z 455.843,A -85,B 0,C 180,E1 -27546.193,E2 -27546.193} C_VEL
LIN {X 0,Y 172.702,Z 467.845,A -85,B 0,C 180,E1 -27547.155,E2 -27547.155} C_VEL
LIN {X 0,Y 165.206,Z 480.39,A -85,B 0,C 180,E1 -27548.488,E2 -27548.488} C_VEL
LIN {X 0,Y 157.057,Z 491.664,A -85,B 0,C 180,E1 -27550.124,E2 -27550.124} C_VEL
LIN {X 0,Y 149.016,Z 501.033,A -85,B 0,C 180,E1 -27551.875,E2 -27551.875} C_VEL
LIN {X 0,Y 139.587,Z 510.371,A -85,B 0,C 180,E1 -27554.262,E2 -27554.262} C_VEL
LIN {X 0,Y 130.445,Z 518.081,A -85,B 0,C 180,E1 -27557.002,E2 -27557.002} C_VEL
LIN {X 0,Y 120.23,Z 525.375,A -85,B 0,C 180,E1 -27560.732,E2 -27560.732} C_VEL
LIN {X 0,Y 111.933,Z 530.39,A -85,B 0,C 180,E1 -27564.441,E2 -27564.441} C_VEL
LIN {X 0,Y 101.789,Z 535.5,A -85,B 0,C 180,E1 -27570.341,E2 -27570.341} C_VEL
LIN {X 0,Y 93.322,Z 538.85,A -85,B 0,C 180,E1 -27577.04,E2 -27577.04} C_VEL
LIN {X 0,Y 87.277,Z 540.598,A -85,B 0,C 180,E1 -27583.556,E2 -27583.556} C_VEL
LIN {X 0,Y 81.447,Z 541.493,A -85,B 0,C 180,E1 -27592.843,E2 -27592.843} C_VEL
LIN {X 0,Y 77.78,Z 540.977,A -85,B 0,C 180,E1 -27603.143,E2 -27603.143} C_VEL
LIN {X 0,Y 76.78,Z 540.195,A -85,B 0,C 180,E1 -27608.524,E2 -27608.524} C_VEL
LIN {X 0,Y 76.29,Z 537.584,A -85,B 0,C 180,E1 -27619.384,E2 -27619.384} C_VEL
LIN {X 0,Y 77.366,Z 534.555,A -85,B 0,C 180,E1 -27627.585,E2 -27627.585} C_VEL
LIN {X 0,Y 79.158,Z 530.883,A -85,B 0,C 180,E1 -27635.094,E2 -27635.094} C_VEL
LIN {X 0,Y 82.029,Z 526.233,A -85,B 0,C 180,E1 -27642.368,E2 -27642.368} C_VEL
LIN {X 0,Y 86.763,Z 519.467,A -85,B 0,C 180,E1 -27650.137,E2 -27650.137} C_VEL
LIN {X 0,Y 92.784,Z 511.049,A -85,B 0,C 180,E1 -27657.031,E2 -27657.031} C_VEL
LIN {X 0,Y 98.832,Z 502.27,A -85,B 0,C 180,E1 -27662.23,E2 -27662.23} C_VEL
LIN {X 0,Y 105.514,Z 491.638,A -85,B 0,C 180,E1 -27666.831,E2 -27666.831} C_VEL
LIN {X 0,Y 111.514,Z 480.902,A -85,B 0,C 180,E1 -27670.24,E2 -27670.24} C_VEL
LIN {X 0,Y 116.368,Z 470.659,A -85,B 0,C 180,E1 -27672.799,E2 -27672.799} C_VEL
LIN {X 0,Y 120.875,Z 459.88,A -85,B 0,C 180,E1 -27674.827,E2 -27674.827} C_VEL
LIN {X 0,Y 125.039,Z 448.478,A -85,B 0,C 180,E1 -27676.356,E2 -27676.356} C_VEL
LIN {X 0,Y 128.815,Z 434.334,A -85,B 0,C 180,E1 -27677.872,E2 -27677.872} C_VEL
LIN {X 0,Y 131.559,Z 420.186,A -85,B 0,C 180,E1 -27678.855,E2 -27678.855} C_VEL
LIN {X 0,Y 133.733,Z 401.044,A -85,B 0,C 180,E1 -27679.644,E2 -27679.644} C_VEL
LIN {X 0,Y 136.501,Z 371.83,A -85,B 0,C 180,E1 -27680.683,E2 -27680.683} C_VEL
LIN {X 0,Y 132.779,Z 363.041,A -85,B 0,C 180,E1 -27684.398,E2 -27684.398} C_VEL
LIN {X 0,Y 129.621,Z 356.624,A -85,B 0,C 180,E1 -27688.013,E2 -27688.013} C_VEL
LIN {X 0,Y 126.625,Z 351.06,A -85,B 0,C 180,E1 -27692.081,E2 -27692.081} C_VEL
LIN {X 0,Y 125.071,Z 348.359,A -85,B 0,C 180,E1 -27694.579,E2 -27694.579} C_VEL
LIN {X 0,Y 123.08,Z 344.963,A -85,B 0,C 180,E1 -27698.47,E2 -27698.47} C_VEL
LIN {X 0,Y 121.163,Z 341.76,A -85,B 0,C 180,E1 -27703.843,E2 -27703.843} C_VEL
LIN {X 0,Y 120.844,Z 340.712,A -85,B 0,C 180,E1 -27705.359,E2 -27705.359} C_VEL
LIN {X 0,Y 119.96,Z 339.868,A -85,B 0,C 180,E1 -27713.276,E2 -27713.276} C_VEL
LIN {X 0,Y 120.948,Z 340.356,A -85,B 0,C 180,E1 -27720.487,E2 -27720.487} C_VEL
LIN {X 0,Y 123.08,Z 344.608,A -85,B 0,C 180,E1 -27727.065,E2 -27727.065} C_VEL
LIN {X 0,Y 125.727,Z 349.475,A -85,B 0,C 180,E1 -27732.139,E2 -27732.139} C_VEL
LIN {X 0,Y 128.287,Z 354.089,A -85,B 0,C 180,E1 -27735.902,E2 -27735.902} C_VEL
LIN {X 0,Y 131.003,Z 359.412,A -85,B 0,C 180,E1 -27739.273,E2 -27739.273} C_VEL
LIN {X 0,Y 134.244,Z 366.516,A -85,B 0,C 180,E1 -27742.767,E2 -27742.767} C_VEL
LIN {X 0,Y 136.434,Z 374.373,A -85,B 0,C 180,E1 -27745.149,E2 -27745.149} C_VEL
LIN {X 0,Y 131.932,Z 420.888,A -85,B 0,C 180,E1 -27746.899,E2 -27746.899} C_VEL
LIN {X 0,Y 129.32,Z 435.243,A -85,B 0,C 180,E1 -27747.76,E2 -27747.76} C_VEL
LIN {X 0,Y 125.885,Z 448.158,A -85,B 0,C 180,E1 -27748.861,E2 -27748.861} C_VEL
LIN {X 0,Y 121.403,Z 461.497,A -85,B 0,C 180,E1 -27750.56,E2 -27750.56} C_VEL
LIN {X 0,Y 116.628,Z 472.883,A -85,B 0,C 180,E1 -27752.475,E2 -27752.475} C_VEL
LIN {X 0,Y 110.962,Z 484.887,A -85,B 0,C 180,E1 -27755.368,E2 -27755.368} C_VEL
LIN {X 0,Y 105.874,Z 493.768,A -85,B 0,C 180,E1 -27757.977,E2 -27757.977} C_VEL
LIN {X 0,Y 100.625,Z 502.316,A -85,B 0,C 180,E1 -27761.34,E2 -27761.34} C_VEL
LIN {X 0,Y 94.184,Z 511.926,A -85,B 0,C 180,E1 -27766.352,E2 -27766.352} C_VEL
LIN {X 0,Y 88.44,Z 520.155,A -85,B 0,C 180,E1 -27772.305,E2 -27772.305} C_VEL
LIN {X 0,Y 83.341,Z 527.481,A -85,B 0,C 180,E1 -27779.604,E2 -27779.604} C_VEL
LIN {X 0,Y 79.995,Z 532.735,A -85,B 0,C 180,E1 -27786.712,E2 -27786.712} C_VEL
LIN {X 0,Y 77.387,Z 538.235,A -85,B 0,C 180,E1 -27796.877,E2 -27796.877} C_VEL
LIN {X 0,Y 76.71,Z 541.25,A -85,B 0,C 180,E1 -27804.743,E2 -27804.743} C_VEL
LIN {X 0,Y 76.853,Z 542.814,A -85,B 0,C 180,E1 -27809.999,E2 -27809.999} C_VEL
LIN {X 0,Y 76.773,Z 543.989,A -85,B 0,C 180,E1 -27815.252,E2 -27815.252} C_VEL
LIN {X 0,Y 77.945,Z 545.325,A -85,B 0,C 180,E1 -27825.693,E2 -27825.693} C_VEL
LIN {X 0,Y 81.301,Z 545.362,A -85,B 0,C 180,E1 -27835.607,E2 -27835.607} C_VEL
LIN {X 0,Y 86.914,Z 544.121,A -85,B 0,C 180,E1 -27844.472,E2 -27844.472} C_VEL
LIN {X 0,Y 94.287,Z 541.579,A -85,B 0,C 180,E1 -27852.13,E2 -27852.13} C_VEL
LIN {X 0,Y 103.127,Z 537.662,A -85,B 0,C 180,E1 -27858.557,E2 -27858.557} C_VEL
LIN {X 0,Y 113.091,Z 532.226,A -85,B 0,C 180,E1 -27863.886,E2 -27863.886} C_VEL
LIN {X 0,Y 121.209,Z 527.087,A -85,B 0,C 180,E1 -27867.216,E2 -27867.216} C_VEL
LIN {X 0,Y 131.159,Z 519.742,A -85,B 0,C 180,E1 -27870.541,E2 -27870.541} C_VEL
LIN {X 0,Y 141.392,Z 510.669,A -85,B 0,C 180,E1 -27873.467,E2 -27873.467} C_VEL
LIN {X 0,Y 150.497,Z 501.211,A -85,B 0,C 180,E1 -27875.588,E2 -27875.588} C_VEL
LIN {X 0,Y 159.058,Z 490.755,A -85,B 0,C 180,E1 -27877.27,E2 -27877.27} C_VEL
LIN {X 0,Y 166.925,Z 479.27,A -85,B 0,C 180,E1 -27878.67,E2 -27878.67} C_VEL
LIN {X 0,Y 171.297,Z 471.893,A -85,B 0,C 180,E1 -27879.347,E2 -27879.347} C_VEL
LIN {X 0,Y 172.977,Z 468.566,A -85,B 0,C 180,E1 -27879.821,E2 -27879.821} C_VEL
LIN {X 0,Y 174.93,Z 463.401,A -85,B 0,C 180,E1 -27881.11,E2 -27881.11} C_VEL
LIN {X 0,Y 176.758,Z 458.103,A -85,B 0,C 180,E1 -27882.341,E2 -27882.341} C_VEL
LIN {X 0,Y 178.11,Z 454.572,A -85,B 0,C 180,E1 -27882.744,E2 -27882.744} C_VEL
LIN {X 0,Y 183.365,Z 440.051,A -85,B 0,C 180,E1 -27883.37,E2 -27883.37} C_VEL
LIN {X 0,Y 187.053,Z 425.812,A -85,B 0,C 180,E1 -27883.771,E2 -27883.771} C_VEL
LIN {X 0,Y 188.053,Z 420.234,A -85,B 0,C 180,E1 -27883.964,E2 -27883.964} C_VEL
LIN {X 0,Y 187.565,Z 417.663,A -85,B 0,C 180,E1 -27885.857,E2 -27885.857} C_VEL
LIN {X 0,Y 186.746,Z 414.808,A -85,B 0,C 180,E1 -27889.7,E2 -27889.7} C_VEL
LIN {X 0,Y 186.429,Z 414.289,A -85,B 0,C 180,E1 -27893.503,E2 -27893.503} C_VEL
LIN {X 0,Y 186.866,Z 414.756,A -85,B 0,C 180,E1 -27897.303,E2 -27897.303} C_VEL
LIN {X 0,Y 187.651,Z 417.816,A -85,B 0,C 180,E1 -27900.936,E2 -27900.936} C_VEL
LIN {X 0,Y 188.071,Z 419.463,A -85,B 0,C 180,E1 -27902.444,E2 -27902.444} C_VEL
LIN {X 0,Y 184.901,Z 433.636,A -85,B 0,C 180,E1 -27902.875,E2 -27902.875} C_VEL
LIN {X 0,Y 180.417,Z 447.533,A -85,B 0,C 180,E1 -27903.464,E2 -27903.464} C_VEL
LIN {X 0,Y 174.852,Z 460.652,A -85,B 0,C 180,E1 -27904.28,E2 -27904.28} C_VEL
LIN {X 0,Y 168.498,Z 472.566,A -85,B 0,C 180,E1 -27905.258,E2 -27905.258} C_VEL
LIN {X 0,Y 160.923,Z 484.223,A -85,B 0,C 180,E1 -27906.519,E2 -27906.519} C_VEL
LIN {X 0,Y 152.655,Z 494.833,A -85,B 0,C 180,E1 -27908.08,E2 -27908.08} C_VEL
LIN {X 0,Y 142.778,Z 505.336,A -85,B 0,C 180,E1 -27910.122,E2 -27910.122} C_VEL
LIN {X 0,Y 132.501,Z 514.481,A -85,B 0,C 180,E1 -27912.68,E2 -27912.68} C_VEL
LIN {X 0,Y 122.311,Z 522.104,A -85,B 0,C 180,E1 -27915.756,E2 -27915.756} C_VEL
LIN {X 0,Y 111.913,Z 528.602,A -85,B 0,C 180,E1 -27919.619,E2 -27919.619} C_VEL
LIN {X 0,Y 101.878,Z 533.789,A -85,B 0,C 180,E1 -27924.444,E2 -27924.444} C_VEL
LIN {X 0,Y 95.669,Z 536.489,A -85,B 0,C 180,E1 -27928.175,E2 -27928.175} C_VEL
LIN {X 0,Y 86.353,Z 539.666,A -85,B 0,C 180,E1 -27935.527,E2 -27935.527} C_VEL
LIN {X 0,Y 78.699,Z 541.366,A -85,B 0,C 180,E1 -27944.407,E2 -27944.407} C_VEL
LIN {X 0,Y 73.105,Z 541.643,A -85,B 0,C 180,E1 -27954.775,E2 -27954.775} C_VEL
LIN {X 0,Y 69.994,Z 540.511,A -85,B 0,C 180,E1 -27966.321,E2 -27966.321} C_VEL
LIN {X 0,Y 69.121,Z 537.991,A -85,B 0,C 180,E1 -27978.268,E2 -27978.268} C_VEL
LIN {X 0,Y 70.306,Z 534.73,A -85,B 0,C 180,E1 -27988.167,E2 -27988.167} C_VEL
LIN {X 0,Y 72.96,Z 530.019,A -85,B 0,C 180,E1 -27998.308,E2 -27998.308} C_VEL
LIN {X 0,Y 76.314,Z 525.103,A -85,B 0,C 180,E1 -28006.039,E2 -28006.039} C_VEL
LIN {X 0,Y 81.81,Z 518.013,A -85,B 0,C 180,E1 -28014.083,E2 -28014.083} C_VEL
LIN {X 0,Y 88.563,Z 509.243,A -85,B 0,C 180,E1 -28021.052,E2 -28021.052} C_VEL
LIN {X 0,Y 95.196,Z 500.06,A -85,B 0,C 180,E1 -28026.2,E2 -28026.2} C_VEL
LIN {X 0,Y 101.408,Z 490.473,A -85,B 0,C 180,E1 -28030.166,E2 -28030.166} C_VEL
LIN {X 0,Y 107.476,Z 479.995,A -85,B 0,C 180,E1 -28033.361,E2 -28033.361} C_VEL
LIN {X 0,Y 112.544,Z 469.534,A -85,B 0,C 180,E1 -28035.9,E2 -28035.9} C_VEL
LIN {X 0,Y 118.059,Z 456.634,A -85,B 0,C 180,E1 -28038.083,E2 -28038.083} C_VEL
LIN {X 0,Y 121.656,Z 446.557,A -85,B 0,C 180,E1 -28039.307,E2 -28039.307} C_VEL
LIN {X 0,Y 125.408,Z 432.44,A -85,B 0,C 180,E1 -28040.719,E2 -28040.719} C_VEL
LIN {X 0,Y 128.117,Z 418.253,A -85,B 0,C 180,E1 -28041.606,E2 -28041.606} C_VEL
LIN {X 0,Y 131.159,Z 390.042,A -85,B 0,C 180,E1 -28042.637,E2 -28042.637} C_VEL
LIN {X 0,Y 132.594,Z 374.619,A -85,B 0,C 180,E1 -28043.236,E2 -28043.236} C_VEL
LIN {X 0,Y 129.096,Z 366.101,A -85,B 0,C 180,E1 -28047.264,E2 -28047.264} C_VEL
LIN {X 0,Y 126.09,Z 359.903,A -85,B 0,C 180,E1 -28051.314,E2 -28051.314} C_VEL
LIN {X 0,Y 123.567,Z 354.982,A -85,B 0,C 180,E1 -28055.505,E2 -28055.505} C_VEL
LIN {X 0,Y 121.599,Z 351.513,A -85,B 0,C 180,E1 -28059.715,E2 -28059.715} C_VEL
LIN {X 0,Y 119.975,Z 348.288,A -85,B 0,C 180,E1 -28065.05,E2 -28065.05} C_VEL
LIN {X 0,Y 119.714,Z 347.606,A -85,B 0,C 180,E1 -28066.423,E2 -28066.423} C_VEL
LIN {X 0,Y 119.081,Z 346.919,A -85,B 0,C 180,E1 -28073.226,E2 -28073.226} C_VEL
LIN {X 0,Y 119.942,Z 347.324,A -85,B 0,C 180,E1 -28080.005,E2 -28080.005} C_VEL
LIN {X 0,Y 121.657,Z 351.233,A -85,B 0,C 180,E1 -28085.952,E2 -28085.952} C_VEL
LIN {X 0,Y 124.036,Z 355.907,A -85,B 0,C 180,E1 -28090.976,E2 -28090.976} C_VEL
LIN {X 0,Y 126.898,Z 361.403,A -85,B 0,C 180,E1 -28095.462,E2 -28095.462} C_VEL
LIN {X 0,Y 130.231,Z 368.931,A -85,B 0,C 180,E1 -28099.765,E2 -28099.765} C_VEL
LIN {X 0,Y 131.488,Z 372.33,A -85,B 0,C 180,E1 -28101.245,E2 -28101.245} C_VEL
LIN {X 0,Y 132.6,Z 376.648,A -85,B 0,C 180,E1 -28102.619,E2 -28102.619} C_VEL
LIN {X 0,Y 128.172,Z 420.686,A -85,B 0,C 180,E1 -28104.25,E2 -28104.25} C_VEL
LIN {X 0,Y 125.428,Z 435.233,A -85,B 0,C 180,E1 -28105.097,E2 -28105.097} C_VEL
LIN {X 0,Y 121.857,Z 448.174,A -85,B 0,C 180,E1 -28106.164,E2 -28106.164} C_VEL
LIN {X 0,Y 117.205,Z 461.466,A -85,B 0,C 180,E1 -28107.816,E2 -28107.816} C_VEL
LIN {X 0,Y 111.718,Z 473.925,A -85,B 0,C 180,E1 -28109.906,E2 -28109.906} C_VEL
LIN {X 0,Y 105.63,Z 485.989,A -85,B 0,C 180,E1 -28112.861,E2 -28112.861} C_VEL
LIN {X 0,Y 100.968,Z 493.66,A -85,B 0,C 180,E1 -28115.128,E2 -28115.128} C_VEL
LIN {X 0,Y 94.832,Z 503.092,A -85,B 0,C 180,E1 -28118.909,E2 -28118.909} C_VEL
LIN {X 0,Y 88.061,Z 512.51,A -85,B 0,C 180,E1 -28124.088,E2 -28124.088} C_VEL
LIN {X 0,Y 82.154,Z 520.344,A -85,B 0,C 180,E1 -28130.092,E2 -28130.092} C_VEL
LIN {X 0,Y 77.244,Z 526.832,A -85,B 0,C 180,E1 -28136.913,E2 -28136.913} C_VEL
LIN {X 0,Y 73.468,Z 532.164,A -85,B 0,C 180,E1 -28144.502,E2 -28144.502} C_VEL
LIN {X 0,Y 70.466,Z 537.763,A -85,B 0,C 180,E1 -28155.561,E2 -28155.561} C_VEL
LIN {X 0,Y 69.622,Z 540.847,A -85,B 0,C 180,E1 -28164.206,E2 -28164.206} C_VEL
LIN {X 0,Y 69.749,Z 542.45,A -85,B 0,C 180,E1 -28169.999,E2 -28169.999} C_VEL
LIN {X 0,Y 69.713,Z 543.662,A -85,B 0,C 180,E1 -28175.785,E2 -28175.785} C_VEL
LIN {X 0,Y 71.116,Z 545.07,A -85,B 0,C 180,E1 -28187.245,E2 -28187.245} C_VEL
LIN {X 0,Y 74.937,Z 545.179,A -85,B 0,C 180,E1 -28197.963,E2 -28197.963} C_VEL
LIN {X 0,Y 81.134,Z 544.011,A -85,B 0,C 180,E1 -28207.325,E2 -28207.325} C_VEL
LIN {X 0,Y 89.126,Z 541.544,A -85,B 0,C 180,E1 -28215.208,E2 -28215.208} C_VEL
LIN {X 0,Y 98.561,Z 537.714,A -85,B 0,C 180,E1 -28221.66,E2 -28221.66} C_VEL
LIN {X 0,Y 109.046,Z 532.392,A -85,B 0,C 180,E1 -28226.911,E2 -28226.911} C_VEL
LIN {X 0,Y 117.523,Z 527.296,A -85,B 0,C 180,E1 -28230.122,E2 -28230.122} C_VEL
LIN {X 0,Y 127.822,Z 520.051,A -85,B 0,C 180,E1 -28233.309,E2 -28233.309} C_VEL
LIN {X 0,Y 138.378,Z 511.152,A -85,B 0,C 180,E1 -28236.087,E2 -28236.087} C_VEL
LIN {X 0,Y 146.134,Z 503.496,A -85,B 0,C 180,E1 -28237.783,E2 -28237.783} C_VEL
LIN {X 0,Y 155.677,Z 492.596,A -85,B 0,C 180,E1 -28239.509,E2 -28239.509} C_VEL
LIN {X 0,Y 163.686,Z 481.56,A -85,B 0,C 180,E1 -28240.832,E2 -28240.832} C_VEL
LIN {X 0,Y 171.035,Z 469.392,A -85,B 0,C 180,E1 -28241.843,E2 -28241.843} C_VEL
LIN {X 0,Y 177.482,Z 456.062,A -85,B 0,C 180,E1 -28242.673,E2 -28242.673} C_VEL
LIN {X 0,Y 178.11,Z 454.572,A -85,B 0,C 180,E1 -28242.744,E2 -28242.744} C_VEL
LIN {X 0,Y 180.141,Z 449.203,A -85,B 0,C 180,E1 -28243.19,E2 -28243.19} C_VEL
LIN {X 0,Y 182.644,Z 440.441,A -85,B 0,C 180,E1 -28244.428,E2 -28244.428} C_VEL
LIN {X 0,Y 184.75,Z 431.497,A -85,B 0,C 180,E1 -28245.576,E2 -28245.576} C_VEL
LIN {X 0,Y 185.969,Z 425.844,A -85,B 0,C 180,E1 -28245.922,E2 -28245.922} C_VEL
LIN {X 0,Y 186.148,Z 424.773,A -85,B 0,C 180,E1 -28246.038,E2 -28246.038} C_VEL
LIN {X 0,Y 185.486,Z 421.739,A -85,B 0,C 180,E1 -28250.098,E2 -28250.098} C_VEL
LIN {X 0,Y 185.247,Z 421.287,A -85,B 0,C 180,E1 -28253.462,E2 -28253.462} C_VEL
LIN {X 0,Y 185.584,Z 421.716,A -85,B 0,C 180,E1 -28257.012,E2 -28257.012} C_VEL
LIN {X 0,Y 186.095,Z 424.519,A -85,B 0,C 180,E1 -28260.414,E2 -28260.414} C_VEL
LIN {X 0,Y 182.381,Z 438.695,A -85,B 0,C 180,E1 -28260.87,E2 -28260.87} C_VEL
LIN {X 0,Y 177.993,Z 450.975,A -85,B 0,C 180,E1 -28261.403,E2 -28261.403} C_VEL
LIN {X 0,Y 172.69,Z 462.694,A -85,B 0,C 180,E1 -28262.105,E2 -28262.105} C_VEL
LIN {X 0,Y 166.259,Z 474.205,A -85,B 0,C 180,E1 -28262.998,E2 -28262.998} C_VEL
LIN {X 0,Y 158.544,Z 485.575,A -85,B 0,C 180,E1 -28264.163,E2 -28264.163} C_VEL
LIN {X 0,Y 149.581,Z 496.535,A -85,B 0,C 180,E1 -28265.7,E2 -28265.7} C_VEL
LIN {X 0,Y 140,Z 506.295,A -85,B 0,C 180,E1 -28267.51,E2 -28267.51} C_VEL
LIN {X 0,Y 130.543,Z 514.452,A -85,B 0,C 180,E1 -28269.639,E2 -28269.639} C_VEL
LIN {X 0,Y 120.502,Z 521.778,A -85,B 0,C 180,E1 -28272.345,E2 -28272.345} C_VEL
LIN {X 0,Y 109.635,Z 528.375,A -85,B 0,C 180,E1 -28275.945,E2 -28275.945} C_VEL
LIN {X 0,Y 100.739,Z 532.886,A -85,B 0,C 180,E1 -28279.651,E2 -28279.651} C_VEL
LIN {X 0,Y 92.362,Z 536.412,A -85,B 0,C 180,E1 -28284.066,E2 -28284.066} C_VEL
LIN {X 0,Y 82.24,Z 539.719,A -85,B 0,C 180,E1 -28291.291,E2 -28291.291} C_VEL
LIN {X 0,Y 73.648,Z 541.509,A -85,B 0,C 180,E1 -28300.237,E2 -28300.237} C_VEL
LIN {X 0,Y 67.15,Z 541.874,A -85,B 0,C 180,E1 -28311.101,E2 -28311.101} C_VEL
LIN {X 0,Y 63.302,Z 540.828,A -85,B 0,C 180,E1 -28323.636,E2 -28323.636} C_VEL
LIN {X 0,Y 62.002,Z 538.393,A -85,B 0,C 180,E1 -28336.898,E2 -28336.898} C_VEL
LIN {X 0,Y 63.451,Z 534.523,A -85,B 0,C 180,E1 -28350.001,E2 -28350.001} C_VEL
LIN {X 0,Y 65.875,Z 530.601,A -85,B 0,C 180,E1 -28359.209,E2 -28359.209} C_VEL
LIN {X 0,Y 69.5,Z 525.783,A -85,B 0,C 180,E1 -28367.66,E2 -28367.66} C_VEL
LIN {X 0,Y 75.37,Z 518.805,A -85,B 0,C 180,E1 -28376.291,E2 -28376.291} C_VEL
LIN {X 0,Y 82.552,Z 510.161,A -85,B 0,C 180,E1 -28383.599,E2 -28383.599} C_VEL
LIN {X 0,Y 89.558,Z 501.123,A -85,B 0,C 180,E1 -28388.887,E2 -28388.887} C_VEL
LIN {X 0,Y 96.049,Z 491.793,A -85,B 0,C 180,E1 -28392.854,E2 -28392.854} C_VEL
LIN {X 0,Y 102.451,Z 481.431,A -85,B 0,C 180,E1 -28396.077,E2 -28396.077} C_VEL
LIN {X 0,Y 107.789,Z 471.219,A -85,B 0,C 180,E1 -28398.573,E2 -28398.573} C_VEL
LIN {X 0,Y 112.687,Z 460.482,A -85,B 0,C 180,E1 -28400.515,E2 -28400.515} C_VEL
LIN {X 0,Y 117.538,Z 448.002,A -85,B 0,C 180,E1 -28402.047,E2 -28402.047} C_VEL
LIN {X 0,Y 121.428,Z 434.322,A -85,B 0,C 180,E1 -28403.422,E2 -28403.422} C_VEL
LIN {X 0,Y 124.401,Z 419.781,A -85,B 0,C 180,E1 -28404.35,E2 -28404.35} C_VEL
LIN {X 0,Y 126.844,Z 399.036,A -85,B 0,C 180,E1 -28405.136,E2 -28405.136} C_VEL
LIN {X 0,Y 128.982,Z 377.692,A -85,B 0,C 180,E1 -28405.888,E2 -28405.888} C_VEL
LIN {X 0,Y 126.125,Z 370.387,A -85,B 0,C 180,E1 -28409.686,E2 -28409.686} C_VEL
LIN {X 0,Y 123.336,Z 364.221,A -85,B 0,C 180,E1 -28414.091,E2 -28414.091} C_VEL
LIN {X 0,Y 121.677,Z 360.972,A -85,B 0,C 180,E1 -28417.289,E2 -28417.289} C_VEL
LIN {X 0,Y 120.346,Z 358.31,A -85,B 0,C 180,E1 -28420.536,E2 -28420.536} C_VEL
LIN {X 0,Y 118.773,Z 354.596,A -85,B 0,C 180,E1 -28426.709,E2 -28426.709} C_VEL
LIN {X 0,Y 118.202,Z 353.969,A -85,B 0,C 180,E1 -28433.175,E2 -28433.175} C_VEL
LIN {X 0,Y 118.932,Z 354.321,A -85,B 0,C 180,E1 -28439.477,E2 -28439.477} C_VEL
LIN {X 0,Y 120.387,Z 357.95,A -85,B 0,C 180,E1 -28445.076,E2 -28445.076} C_VEL
LIN {X 0,Y 122.459,Z 362.49,A -85,B 0,C 180,E1 -28449.918,E2 -28449.918} C_VEL
LIN {X 0,Y 124.94,Z 367.66,A -85,B 0,C 180,E1 -28454.173,E2 -28454.173} C_VEL
LIN {X 0,Y 127.8,Z 374.698,A -85,B 0,C 180,E1 -28458.256,E2 -28458.256} C_VEL
LIN {X 0,Y 128.662,Z 377.479,A -85,B 0,C 180,E1 -28459.424,E2 -28459.424} C_VEL
LIN {X 0,Y 129.029,Z 379.022,A -85,B 0,C 180,E1 -28459.946,E2 -28459.946} C_VEL
LIN {X 0,Y 124.752,Z 420.212,A -85,B 0,C 180,E1 -28461.44,E2 -28461.44} C_VEL
LIN {X 0,Y 121.893,Z 434.927,A -85,B 0,C 180,E1 -28462.246,E2 -28462.246} C_VEL
LIN {X 0,Y 118.117,Z 448.19,A -85,B 0,C 180,E1 -28463.289,E2 -28463.289} C_VEL
LIN {X 0,Y 113.295,Z 461.436,A -85,B 0,C 180,E1 -28464.877,E2 -28464.877} C_VEL
LIN {X 0,Y 107.552,Z 473.954,A -85,B 0,C 180,E1 -28466.908,E2 -28466.908} C_VEL
LIN {X 0,Y 101.223,Z 485.903,A -85,B 0,C 180,E1 -28469.788,E2 -28469.788} C_VEL
LIN {X 0,Y 96.344,Z 493.555,A -85,B 0,C 180,E1 -28472.005,E2 -28472.005} C_VEL
LIN {X 0,Y 90.509,Z 502.091,A -85,B 0,C 180,E1 -28475.381,E2 -28475.381} C_VEL
LIN {X 0,Y 83.206,Z 511.666,A -85,B 0,C 180,E1 -28480.52,E2 -28480.52} C_VEL
LIN {X 0,Y 76.598,Z 519.846,A -85,B 0,C 180,E1 -28486.879,E2 -28486.879} C_VEL
LIN {X 0,Y 71.343,Z 526.169,A -85,B 0,C 180,E1 -28493.768,E2 -28493.768} C_VEL
LIN {X 0,Y 67.075,Z 531.594,A -85,B 0,C 180,E1 -28501.868,E2 -28501.868} C_VEL
LIN {X 0,Y 63.554,Z 537.278,A -85,B 0,C 180,E1 -28513.951,E2 -28513.951} C_VEL
LIN {X 0,Y 62.552,Z 540.444,A -85,B 0,C 180,E1 -28523.548,E2 -28523.548} C_VEL
LIN {X 0,Y 62.644,Z 542.086,A -85,B 0,C 180,E1 -28529.999,E2 -28529.999} C_VEL
LIN {X 0,Y 62.634,Z 543.334,A -85,B 0,C 180,E1 -28536.442,E2 -28536.442} C_VEL
LIN {X 0,Y 64.338,Z 544.814,A -85,B 0,C 180,E1 -28549.128,E2 -28549.128} C_VEL
LIN {X 0,Y 68.728,Z 544.997,A -85,B 0,C 180,E1 -28560.748,E2 -28560.748} C_VEL
LIN {X 0,Y 75.587,Z 543.902,A -85,B 0,C 180,E1 -28570.604,E2 -28570.604} C_VEL
LIN {X 0,Y 84.255,Z 541.508,A -85,B 0,C 180,E1 -28578.651,E2 -28578.651} C_VEL
LIN {X 0,Y 94.299,Z 537.756,A -85,B 0,C 180,E1 -28585.064,E2 -28585.064} C_VEL
LIN {X 0,Y 105.329,Z 532.544,A -85,B 0,C 180,E1 -28590.157,E2 -28590.157} C_VEL
LIN {X 0,Y 114.159,Z 527.521,A -85,B 0,C 180,E1 -28593.207,E2 -28593.207} C_VEL
LIN {X 0,Y 124.8,Z 520.385,A -85,B 0,C 180,E1 -28596.216,E2 -28596.216} C_VEL
LIN {X 0,Y 135.667,Z 511.614,A -85,B 0,C 180,E1 -28598.817,E2 -28598.817} C_VEL
LIN {X 0,Y 145.238,Z 502.453,A -85,B 0,C 180,E1 -28600.66,E2 -28600.66} C_VEL
LIN {X 0,Y 153.355,Z 493.325,A -85,B 0,C 180,E1 -28601.973,E2 -28601.973} C_VEL
LIN {X 0,Y 161.514,Z 482.483,A -85,B 0,C 180,E1 -28603.189,E2 -28603.189} C_VEL
LIN {X 0,Y 168.974,Z 470.609,A -85,B 0,C 180,E1 -28604.111,E2 -28604.111} C_VEL
LIN {X 0,Y 175.553,Z 457.663,A -85,B 0,C 180,E1 -28604.857,E2 -28604.857} C_VEL
LIN {X 0,Y 181.14,Z 443.35,A -85,B 0,C 180,E1 -28605.461,E2 -28605.461} C_VEL
LIN {X 0,Y 185.278,Z 428.791,A -85,B 0,C 180,E1 -28605.869,E2 -28605.869} C_VEL
LIN {X 0,Y 185.969,Z 425.844,A -85,B 0,C 180,E1 -28605.922,E2 -28605.922} C_VEL
LIN {X 0,Y 186.238,Z 424.272,A -85,B 0,C 180,E1 -28606.169,E2 -28606.169} C_VEL
LIN {X 0,Y 186.268,Z 422.752,A -85,B 0,C 180,E1 -28606.995,E2 -28606.995} C_VEL
LIN {X 0,Y 186.04,Z 422.333,A -85,B 0,C 180,E1 -28607.93,E2 -28607.93} C_VEL
LIN {X 0,Y 185.647,Z 422.585,A -85,B 0,C 180,E1 -28609.081,E2 -28609.081} C_VEL
LIN {X 0,Y 183.884,Z 427.837,A -85,B 0,C 180,E1 -28614.583,E2 -28614.583} C_VEL
LIN {X 0,Y 183.9,Z 428.299,A -85,B 0,C 180,E1 -28615.766,E2 -28615.766} C_VEL
LIN {X 0,Y 183.987,Z 428.714,A -85,B 0,C 180,E1 -28616.849,E2 -28616.849} C_VEL
LIN {X 0,Y 184.084,Z 429.836,A -85,B 0,C 180,E1 -28618.349,E2 -28618.349} C_VEL
LIN {X 0,Y 180.1,Z 443.207,A -85,B 0,C 180,E1 -28618.784,E2 -28618.784} C_VEL
LIN {X 0,Y 174.826,Z 456.396,A -85,B 0,C 180,E1 -28619.372,E2 -28619.372} C_VEL
LIN {X 0,Y 168.668,Z 468.501,A -85,B 0,C 180,E1 -28620.114,E2 -28620.114} C_VEL
LIN {X 0,Y 160.793,Z 480.961,A -85,B 0,C 180,E1 -28621.136,E2 -28621.136} C_VEL
LIN {X 0,Y 151.944,Z 492.423,A -85,B 0,C 180,E1 -28622.406,E2 -28622.406} C_VEL
LIN {X 0,Y 142.642,Z 502.439,A -85,B 0,C 180,E1 -28623.895,E2 -28623.895} C_VEL
LIN {X 0,Y 131.857,Z 512.112,A -85,B 0,C 180,E1 -28625.897,E2 -28625.897} C_VEL
LIN {X 0,Y 120.772,Z 520.36,A -85,B 0,C 180,E1 -28628.414,E2 -28628.414} C_VEL
LIN {X 0,Y 109.832,Z 527.082,A -85,B 0,C 180,E1 -28631.487,E2 -28631.487} C_VEL
LIN {X 0,Y 98.48,Z 532.762,A -85,B 0,C 180,E1 -28635.551,E2 -28635.551} C_VEL
LIN {X 0,Y 89.573,Z 536.338,A -85,B 0,C 180,E1 -28639.694,E2 -28639.694} C_VEL
LIN {X 0,Y 78.608,Z 539.756,A -85,B 0,C 180,E1 -28646.617,E2 -28646.617} C_VEL
LIN {X 0,Y 69.041,Z 541.652,A -85,B 0,C 180,E1 -28655.479,E2 -28655.479} C_VEL
LIN {X 0,Y 61.538,Z 542.105,A -85,B 0,C 180,E1 -28666.748,E2 -28666.748} C_VEL
LIN {X 0,Y 56.764,Z 541.147,A -85,B 0,C 180,E1 -28680.316,E2 -28680.316} C_VEL
LIN {X 0,Y 54.917,Z 538.795,A -85,B 0,C 180,E1 -28695.171,E2 -28695.171} C_VEL
LIN {X 0,Y 56.254,Z 535.01,A -85,B 0,C 180,E1 -28710.001,E2 -28710.001} C_VEL
LIN {X 0,Y 58.818,Z 531.182,A -85,B 0,C 180,E1 -28720.326,E2 -28720.326} C_VEL
LIN {X 0,Y 62.759,Z 526.462,A -85,B 0,C 180,E1 -28729.631,E2 -28729.631} C_VEL
LIN {X 0,Y 69.066,Z 519.597,A -85,B 0,C 180,E1 -28738.904,E2 -28738.904} C_VEL
LIN {X 0,Y 75.569,Z 512.439,A -85,B 0,C 180,E1 -28745.539,E2 -28745.539} C_VEL
LIN {X 0,Y 82.87,Z 503.819,A -85,B 0,C 180,E1 -28751.091,E2 -28751.091} C_VEL
LIN {X 0,Y 90.212,Z 494.171,A -85,B 0,C 180,E1 -28755.45,E2 -28755.45} C_VEL
LIN {X 0,Y 95.6,Z 486.214,A -85,B 0,C 180,E1 -28758.102,E2 -28758.102} C_VEL
LIN {X 0,Y 102.607,Z 474.226,A -85,B 0,C 180,E1 -28761.18,E2 -28761.18} C_VEL
LIN {X 0,Y 107.562,Z 464.041,A -85,B 0,C 180,E1 -28763.167,E2 -28763.167} C_VEL
LIN {X 0,Y 112.215,Z 453.398,A -85,B 0,C 180,E1 -28764.506,E2 -28764.506} C_VEL
LIN {X 0,Y 116.63,Z 440.118,A -85,B 0,C 180,E1 -28765.95,E2 -28765.95} C_VEL
LIN {X 0,Y 120.162,Z 425.718,A -85,B 0,C 180,E1 -28767.011,E2 -28767.011} C_VEL
LIN {X 0,Y 122.442,Z 411.384,A -85,B 0,C 180,E1 -28767.658,E2 -28767.658} C_VEL
LIN {X 0,Y 125.627,Z 381.69,A -85,B 0,C 180,E1 -28768.589,E2 -28768.589} C_VEL
LIN {X 0,Y 125.552,Z 380.606,A -85,B 0,C 180,E1 -28768.822,E2 -28768.822} C_VEL
LIN {X 0,Y 123.483,Z 375.094,A -85,B 0,C 180,E1 -28772.015,E2 -28772.015} C_VEL
LIN {X 0,Y 121.269,Z 369.795,A -85,B 0,C 180,E1 -28776.072,E2 -28776.072} C_VEL
LIN {X 0,Y 119.931,Z 366.991,A -85,B 0,C 180,E1 -28779.074,E2 -28779.074} C_VEL
LIN {X 0,Y 118.999,Z 364.915,A -85,B 0,C 180,E1 -28781.725,E2 -28781.725} C_VEL
LIN {X 0,Y 117.763,Z 361.555,A -85,B 0,C 180,E1 -28787.387,E2 -28787.387} C_VEL
LIN {X 0,Y 117.327,Z 360.994,A -85,B 0,C 180,E1 -28793.124,E2 -28793.124} C_VEL
LIN {X 0,Y 117.904,Z 361.257,A -85,B 0,C 180,E1 -28798.771,E2 -28798.771} C_VEL
LIN {X 0,Y 119.38,Z 365.395,A -85,B 0,C 180,E1 -28804.948,E2 -28804.948} C_VEL
LIN {X 0,Y 120.861,Z 368.896,A -85,B 0,C 180,E1 -28808.688,E2 -28808.688} C_VEL
LIN {X 0,Y 123.196,Z 374.26,A -85,B 0,C 180,E1 -28813.106,E2 -28813.106} C_VEL
LIN {X 0,Y 125.679,Z 381.138,A -85,B 0,C 180,E1 -28817.017,E2 -28817.017} C_VEL
LIN {X 0,Y 125.766,Z 381.551,A -85,B 0,C 180,E1 -28817.165,E2 -28817.165} C_VEL
LIN {X 0,Y 121.498,Z 420.618,A -85,B 0,C 180,E1 -28818.516,E2 -28818.516} C_VEL
LIN {X 0,Y 118.632,Z 434.782,A -85,B 0,C 180,E1 -28819.239,E2 -28819.239} C_VEL
LIN {X 0,Y 114.694,Z 448.206,A -85,B 0,C 180,E1 -28820.236,E2 -28820.236} C_VEL
LIN {X 0,Y 109.705,Z 461.405,A -85,B 0,C 180,E1 -28821.737,E2 -28821.737} C_VEL
LIN {X 0,Y 103.616,Z 474.147,A -85,B 0,C 180,E1 -28823.706,E2 -28823.706} C_VEL
LIN {X 0,Y 97.134,Z 485.818,A -85,B 0,C 180,E1 -28826.445,E2 -28826.445} C_VEL
LIN {X 0,Y 92.035,Z 493.45,A -85,B 0,C 180,E1 -28828.579,E2 -28828.579} C_VEL
LIN {X 0,Y 85.203,Z 502.855,A -85,B 0,C 180,E1 -28832.278,E2 -28832.278} C_VEL
LIN {X 0,Y 77.511,Z 512.24,A -85,B 0,C 180,E1 -28837.499,E2 -28837.499} C_VEL
LIN {X 0,Y 70.66,Z 520.053,A -85,B 0,C 180,E1 -28843.855,E2 -28843.855} C_VEL
LIN {X 0,Y 63.929,Z 527.477,A -85,B 0,C 180,E1 -28852.797,E2 -28852.797} C_VEL
LIN {X 0,Y 59.512,Z 532.657,A -85,B 0,C 180,E1 -28861.811,E2 -28861.811} C_VEL
LIN {X 0,Y 56.707,Z 536.793,A -85,B 0,C 180,E1 -28871.95,E2 -28871.95} C_VEL
LIN {X 0,Y 55.51,Z 540.043,A -85,B 0,C 180,E1 -28882.726,E2 -28882.726} C_VEL
LIN {X 0,Y 55.534,Z 541.721,A -85,B 0,C 180,E1 -28889.999,E2 -28889.999} C_VEL
LIN {X 0,Y 55.57,Z 543.006,A -85,B 0,C 180,E1 -28897.265,E2 -28897.265} C_VEL
LIN {X 0,Y 57.633,Z 544.558,A -85,B 0,C 180,E1 -28911.458,E2 -28911.458} C_VEL
LIN {X 0,Y 62.714,Z 544.815,A -85,B 0,C 180,E1 -28924.076,E2 -28924.076} C_VEL
LIN {X 0,Y 70.328,Z 543.792,A -85,B 0,C 180,E1 -28934.386,E2 -28934.386} C_VEL
LIN {X 0,Y 79.713,Z 541.477,A -85,B 0,C 180,E1 -28942.511,E2 -28942.511} C_VEL
LIN {X 0,Y 90.409,Z 537.81,A -85,B 0,C 180,E1 -28948.767,E2 -28948.767} C_VEL
LIN {X 0,Y 101.973,Z 532.686,A -85,B 0,C 180,E1 -28953.629,E2 -28953.629} C_VEL
LIN {X 0,Y 111.14,Z 527.754,A -85,B 0,C 180,E1 -28956.476,E2 -28956.476} C_VEL
LIN {X 0,Y 122.107,Z 520.72,A -85,B 0,C 180,E1 -28959.269,E2 -28959.269} C_VEL
LIN {X 0,Y 133.272,Z 512.062,A -85,B 0,C 180,E1 -28961.656,E2 -28961.656} C_VEL
LIN {X 0,Y 143.053,Z 503.03,A -85,B 0,C 180,E1 -28963.331,E2 -28963.331} C_VEL
LIN {X 0,Y 152.98,Z 492.118,A -85,B 0,C 180,E1 -28964.736,E2 -28964.736} C_VEL
LIN {X 0,Y 161.298,Z 481.059,A -85,B 0,C 180,E1 -28965.799,E2 -28965.799} C_VEL
LIN {X 0,Y 168.874,Z 468.862,A -85,B 0,C 180,E1 -28966.597,E2 -28966.597} C_VEL
LIN {X 0,Y 175.382,Z 455.798,A -85,B 0,C 180,E1 -28967.236,E2 -28967.236} C_VEL
LIN {X 0,Y 180.456,Z 442.743,A -85,B 0,C 180,E1 -28967.708,E2 -28967.708} C_VEL
LIN {X 0,Y 184.103,Z 430.242,A -85,B 0,C 180,E1 -28968.067,E2 -28968.067} C_VEL
LIN {X 0,Y 183.92,Z 428.602,A -85,B 0,C 180,E1 -28970.457,E2 -28970.457} C_VEL
LIN {X 0,Y 183.885,Z 428.274,A -85,B 0,C 180,E1 -28975.613,E2 -28975.613} C_VEL
LIN {X 0,Y 183.9,Z 428.299,A -85,B 0,C 180,E1 -28975.766,E2 -28975.766} C_VEL
LIN {X 0,Y 183.777,Z 429.256,A -85,B 0,C 180,E1 -28976.392,E2 -28976.392} C_VEL
LIN {X 0,Y 183.387,Z 431.139,A -85,B 0,C 180,E1 -28976.817,E2 -28976.817} C_VEL
LIN {X 0,Y 182.416,Z 434.779,A -85,B 0,C 180,E1 -28977.116,E2 -28977.116} C_VEL
LIN {X 0,Y 181.027,Z 439.168,A -85,B 0,C 180,E1 -28976.999,E2 -28976.999} C_VEL
LIN {X 0,Y 178.203,Z 446.914,A -85,B 0,C 180,E1 -28976.679,E2 -28976.679} C_VEL
LIN {X 0,Y 177.612,Z 448.432,A -85,B 0,C 180,E1 -28976.708,E2 -28976.708} C_VEL
LIN {X 0,Y 172.38,Z 460.267,A -85,B 0,C 180,E1 -28977.249,E2 -28977.249} C_VEL
LIN {X 0,Y 166.03,Z 471.837,A -85,B 0,C 180,E1 -28977.909,E2 -28977.909} C_VEL
LIN {X 0,Y 158.16,Z 483.572,A -85,B 0,C 180,E1 -28978.802,E2 -28978.802} C_VEL
LIN {X 0,Y 149.045,Z 494.782,A -85,B 0,C 180,E1 -28979.996,E2 -28979.996} C_VEL
LIN {X 0,Y 138.843,Z 505.14,A -85,B 0,C 180,E1 -28981.441,E2 -28981.441} C_VEL
LIN {X 0,Y 128.795,Z 513.63,A -85,B 0,C 180,E1 -28983.124,E2 -28983.124} C_VEL
LIN {X 0,Y 118.215,Z 521.121,A -85,B 0,C 180,E1 -28985.268,E2 -28985.268} C_VEL
LIN {X 0,Y 106.506,Z 527.939,A -85,B 0,C 180,E1 -28988.201,E2 -28988.201} C_VEL
LIN {X 0,Y 96.743,Z 532.607,A -85,B 0,C 180,E1 -28991.278,E2 -28991.278} C_VEL
LIN {X 0,Y 87.331,Z 536.265,A -85,B 0,C 180,E1 -28995.055,E2 -28995.055} C_VEL
LIN {X 0,Y 75.532,Z 539.774,A -85,B 0,C 180,E1 -29001.498,E2 -29001.498} C_VEL
LIN {X 0,Y 64.987,Z 541.786,A -85,B 0,C 180,E1 -29010.103,E2 -29010.103} C_VEL
LIN {X 0,Y 56.337,Z 542.336,A -85,B 0,C 180,E1 -29021.543,E2 -29021.543} C_VEL
LIN {X 0,Y 50.453,Z 541.464,A -85,B 0,C 180,E1 -29036.14,E2 -29036.14} C_VEL
LIN {X 0,Y 47.871,Z 539.198,A -85,B 0,C 180,E1 -29052.927,E2 -29052.927} C_VEL
LIN {X 0,Y 48.996,Z 535.502,A -85,B 0,C 180,E1 -29070.001,E2 -29070.001} C_VEL
LIN {X 0,Y 51.793,Z 531.763,A -85,B 0,C 180,E1 -29081.745,E2 -29081.745} C_VEL
LIN {X 0,Y 56.114,Z 527.125,A -85,B 0,C 180,E1 -29092.07,E2 -29092.07} C_VEL
LIN {X 0,Y 62.923,Z 520.387,A -85,B 0,C 180,E1 -29102.042,E2 -29102.042} C_VEL
LIN {X 0,Y 71.143,Z 511.996,A -85,B 0,C 180,E1 -29109.95,E2 -29109.95} C_VEL
LIN {X 0,Y 78.996,Z 503.247,A -85,B 0,C 180,E1 -29115.376,E2 -29115.376} C_VEL
LIN {X 0,Y 86.77,Z 493.479,A -85,B 0,C 180,E1 -29119.535,E2 -29119.535} C_VEL
LIN {X 0,Y 93.204,Z 484.294,A -85,B 0,C 180,E1 -29122.348,E2 -29122.348} C_VEL
LIN {X 0,Y 100.486,Z 471.762,A -85,B 0,C 180,E1 -29125.264,E2 -29125.264} C_VEL
LIN {X 0,Y 105.775,Z 461.058,A -85,B 0,C 180,E1 -29127.017,E2 -29127.017} C_VEL
LIN {X 0,Y 110.951,Z 448.619,A -85,B 0,C 180,E1 -29128.338,E2 -29128.338} C_VEL
LIN {X 0,Y 115.193,Z 434.732,A -85,B 0,C 180,E1 -29129.595,E2 -29129.595} C_VEL
LIN {X 0,Y 118.398,Z 419.999,A -85,B 0,C 180,E1 -29130.416,E2 -29130.416} C_VEL
LIN {X 0,Y 121.074,Z 398.581,A -85,B 0,C 180,E1 -29131.125,E2 -29131.125} C_VEL
LIN {X 0,Y 122.645,Z 384.354,A -85,B 0,C 180,E1 -29131.528,E2 -29131.528} C_VEL
LIN {X 0,Y 120.56,Z 378.473,A -85,B 0,C 180,E1 -29135.411,E2 -29135.411} C_VEL
LIN {X 0,Y 118.837,Z 374.134,A -85,B 0,C 180,E1 -29139.434,E2 -29139.434} C_VEL
LIN {X 0,Y 117.784,Z 371.612,A -85,B 0,C 180,E1 -29142.685,E2 -29142.685} C_VEL
LIN {X 0,Y 116.818,Z 368.664,A -85,B 0,C 180,E1 -29147.684,E2 -29147.684} C_VEL
LIN {X 0,Y 116.45,Z 368.028,A -85,B 0,C 180,E1 -29153.072,E2 -29153.072} C_VEL
LIN {X 0,Y 116.914,Z 368.357,A -85,B 0,C 180,E1 -29158.268,E2 -29158.268} C_VEL
LIN {X 0,Y 118.083,Z 371.978,A -85,B 0,C 180,E1 -29163.852,E2 -29163.852} C_VEL
LIN {X 0,Y 119.654,Z 376.186,A -85,B 0,C 180,E1 -29168.236,E2 -29168.236} C_VEL
LIN {X 0,Y 121.438,Z 380.844,A -85,B 0,C 180,E1 -29171.931,E2 -29171.931} C_VEL
LIN {X 0,Y 122.725,Z 384.723,A -85,B 0,C 180,E1 -29174.249,E2 -29174.249} C_VEL
LIN {X 0,Y 118.607,Z 420.791,A -85,B 0,C 180,E1 -29175.424,E2 -29175.424} C_VEL
LIN {X 0,Y 115.657,Z 434.856,A -85,B 0,C 180,E1 -29176.087,E2 -29176.087} C_VEL
LIN {X 0,Y 112.027,Z 447.088,A -85,B 0,C 180,E1 -29176.924,E2 -29176.924} C_VEL
LIN {X 0,Y 107.253,Z 459.584,A -85,B 0,C 180,E1 -29178.17,E2 -29178.17} C_VEL
LIN {X 0,Y 101.742,Z 471.195,A -85,B 0,C 180,E1 -29179.753,E2 -29179.753} C_VEL
LIN {X 0,Y 95.674,Z 482.078,A -85,B 0,C 180,E1 -29181.9,E2 -29181.9} C_VEL
LIN {X 0,Y 90.291,Z 490.161,A -85,B 0,C 180,E1 -29183.854,E2 -29183.854} C_VEL
LIN {X 0,Y 83.036,Z 500.056,A -85,B 0,C 180,E1 -29187.291,E2 -29187.291} C_VEL
LIN {X 0,Y 74.696,Z 509.906,A -85,B 0,C 180,E1 -29192.136,E2 -29192.136} C_VEL
LIN {X 0,Y 67.066,Z 518.065,A -85,B 0,C 180,E1 -29198.193,E2 -29198.193} C_VEL
LIN {X 0,Y 60.336,Z 524.838,A -85,B 0,C 180,E1 -29205.663,E2 -29205.663} C_VEL
LIN {X 0,Y 54.876,Z 530.455,A -85,B 0,C 180,E1 -29214.808,E2 -29214.808} C_VEL
LIN {X 0,Y 49.961,Z 536.308,A -85,B 0,C 180,E1 -29229.41,E2 -29229.41} C_VEL
LIN {X 0,Y 48.467,Z 539.64,A -85,B 0,C 180,E1 -29241.662,E2 -29241.662} C_VEL
LIN {X 0,Y 48.445,Z 541.357,A -85,B 0,C 180,E1 -29249.999,E2 -29249.999} C_VEL
LIN {X 0,Y 48.537,Z 542.679,A -85,B 0,C 180,E1 -29258.324,E2 -29258.324} C_VEL
LIN {X 0,Y 51.053,Z 544.302,A -85,B 0,C 180,E1 -29274.391,E2 -29274.391} C_VEL
LIN {X 0,Y 56.935,Z 544.632,A -85,B 0,C 180,E1 -29288.11,E2 -29288.11} C_VEL
LIN {X 0,Y 65.412,Z 543.687,A -85,B 0,C 180,E1 -29298.769,E2 -29298.769} C_VEL
LIN {X 0,Y 75.576,Z 541.45,A -85,B 0,C 180,E1 -29306.814,E2 -29306.814} C_VEL
LIN {X 0,Y 86.934,Z 537.865,A -85,B 0,C 180,E1 -29312.778,E2 -29312.778} C_VEL
LIN {X 0,Y 99.016,Z 532.827,A -85,B 0,C 180,E1 -29317.322,E2 -29317.322} C_VEL
LIN {X 0,Y 111.703,Z 526.183,A -85,B 0,C 180,E1 -29320.687,E2 -29320.687} C_VEL
LIN {X 0,Y 123.021,Z 518.83,A -85,B 0,C 180,E1 -29323.112,E2 -29323.112} C_VEL
LIN {X 0,Y 134.511,Z 509.74,A -85,B 0,C 180,E1 -29325.143,E2 -29325.143} C_VEL
LIN {X 0,Y 144.547,Z 500.257,A -85,B 0,C 180,E1 -29326.505,E2 -29326.505} C_VEL
LIN {X 0,Y 153.814,Z 489.781,A -85,B 0,C 180,E1 -29327.589,E2 -29327.589} C_VEL
LIN {X 0,Y 162.259,Z 478.263,A -85,B 0,C 180,E1 -29328.505,E2 -29328.505} C_VEL
LIN {X 0,Y 169.944,Z 465.463,A -85,B 0,C 180,E1 -29329.158,E2 -29329.158} C_VEL
LIN {X 0,Y 176.123,Z 452.523,A -85,B 0,C 180,E1 -29329.66,E2 -29329.66} C_VEL
LIN {X 0,Y 181.133,Z 438.897,A -85,B 0,C 180,E1 -29330.048,E2 -29330.048} C_VEL
LIN {X 0,Y 182.061,Z 435.715,A -85,B 0,C 180,E1 -29330.174,E2 -29330.174} C_VEL
LIN {X 0,Y 181.907,Z 435.087,A -85,B 0,C 180,E1 -29333.341,E2 -29333.341} C_VEL
LIN {X 0,Y 182.086,Z 435.324,A -85,B 0,C 180,E1 -29336.298,E2 -29336.298} C_VEL
LIN {X 0,Y 177.612,Z 448.432,A -85,B 0,C 180,E1 -29336.708,E2 -29336.708} C_VEL
LIN {X 0,Y 175.349,Z 453.902,A -85,B 0,C 180,E1 -29336.705,E2 -29336.705} C_VEL
LIN {X 0,Y 171.049,Z 462.7,A -85,B 0,C 180,E1 -29336.159,E2 -29336.159} C_VEL
LIN {X 0,Y 166.168,Z 471.168,A -85,B 0,C 180,E1 -29335.644,E2 -29335.644} C_VEL
LIN {X 0,Y 162.974,Z 476.113,A -85,B 0,C 180,E1 -29335.717,E2 -29335.717} C_VEL
LIN {X 0,Y 154.002,Z 488.355,A -85,B 0,C 180,E1 -29336.605,E2 -29336.605} C_VEL
LIN {X 0,Y 144.182,Z 499.346,A -85,B 0,C 180,E1 -29337.745,E2 -29337.745} C_VEL
LIN {X 0,Y 133.545,Z 509.169,A -85,B 0,C 180,E1 -29339.091,E2 -29339.091} C_VEL
LIN {X 0,Y 122.996,Z 517.254,A -85,B 0,C 180,E1 -29340.719,E2 -29340.719} C_VEL
LIN {X 0,Y 112.568,Z 523.915,A -85,B 0,C 180,E1 -29342.678,E2 -29342.678} C_VEL
LIN {X 0,Y 102.296,Z 529.377,A -85,B 0,C 180,E1 -29345.025,E2 -29345.025} C_VEL
LIN {X 0,Y 92.239,Z 533.796,A -85,B 0,C 180,E1 -29347.911,E2 -29347.911} C_VEL
LIN {X 0,Y 79.301,Z 538.185,A -85,B 0,C 180,E1 -29352.883,E2 -29352.883} C_VEL
LIN {X 0,Y 67.186,Z 541.024,A -85,B 0,C 180,E1 -29359.711,E2 -29359.711} C_VEL
LIN {X 0,Y 56.371,Z 542.402,A -85,B 0,C 180,E1 -29369.227,E2 -29369.227} C_VEL
LIN {X 0,Y 47.665,Z 542.347,A -85,B 0,C 180,E1 -29382.508,E2 -29382.508} C_VEL
LIN {X 0,Y 42.182,Z 540.86,A -85,B 0,C 180,E1 -29400.013,E2 -29400.013} C_VEL
LIN {X 0,Y 40.77,Z 537.969,A -85,B 0,C 180,E1 -29420.075,E2 -29420.075} C_VEL
LIN {X 0,Y 42.2,Z 535.39,A -85,B 0,C 180,E1 -29432.567,E2 -29432.567} C_VEL
LIN {X 0,Y 46.224,Z 530.884,A -85,B 0,C 180,E1 -29447.704,E2 -29447.704} C_VEL
LIN {X 0,Y 51.524,Z 525.977,A -85,B 0,C 180,E1 -29458.517,E2 -29458.517} C_VEL
LIN {X 0,Y 59.416,Z 518.909,A -85,B 0,C 180,E1 -29468.389,E2 -29468.389} C_VEL
LIN {X 0,Y 68.568,Z 510.156,A -85,B 0,C 180,E1 -29475.846,E2 -29475.846} C_VEL
LIN {X 0,Y 77.076,Z 500.996,A -85,B 0,C 180,E1 -29480.81,E2 -29480.81} C_VEL
LIN {X 0,Y 85.105,Z 491.002,A -85,B 0,C 180,E1 -29484.532,E2 -29484.532} C_VEL
LIN {X 0,Y 92.082,Z 480.984,A -85,B 0,C 180,E1 -29487.093,E2 -29487.093} C_VEL
LIN {X 0,Y 98.923,Z 469.137,A -85,B 0,C 180,E1 -29489.476,E2 -29489.476} C_VEL
LIN {X 0,Y 105.331,Z 455.92,A -85,B 0,C 180,E1 -29491.131,E2 -29491.131} C_VEL
LIN {X 0,Y 109.763,Z 444.35,A -85,B 0,C 180,E1 -29492.176,E2 -29492.176} C_VEL
LIN {X 0,Y 113.719,Z 430.624,A -85,B 0,C 180,E1 -29493.176,E2 -29493.176} C_VEL
LIN {X 0,Y 116.514,Z 416.572,A -85,B 0,C 180,E1 -29493.779,E2 -29493.779} C_VEL
LIN {X 0,Y 119.864,Z 387.781,A -85,B 0,C 180,E1 -29494.625,E2 -29494.625} C_VEL
LIN {X 0,Y 118.16,Z 382.622,A -85,B 0,C 180,E1 -29498.608,E2 -29498.608} C_VEL
LIN {X 0,Y 117.045,Z 379.625,A -85,B 0,C 180,E1 -29501.94,E2 -29501.94} C_VEL
LIN {X 0,Y 116.431,Z 377.95,A -85,B 0,C 180,E1 -29504.369,E2 -29504.369} C_VEL
LIN {X 0,Y 115.817,Z 375.552,A -85,B 0,C 180,E1 -29508.547,E2 -29508.547} C_VEL
LIN {X 0,Y 115.573,Z 375.065,A -85,B 0,C 180,E1 -29513.019,E2 -29513.019} C_VEL
LIN {X 0,Y 115.938,Z 375.422,A -85,B 0,C 180,E1 -29517.761,E2 -29517.761} C_VEL
LIN {X 0,Y 116.863,Z 378.776,A -85,B 0,C 180,E1 -29522.905,E2 -29522.905} C_VEL
LIN {X 0,Y 118.131,Z 382.582,A -85,B 0,C 180,E1 -29526.945,E2 -29526.945} C_VEL
LIN {X 0,Y 119.568,Z 386.894,A -85,B 0,C 180,E1 -29530.375,E2 -29530.375} C_VEL
LIN {X 0,Y 119.925,Z 388.101,A -85,B 0,C 180,E1 -29531.144,E2 -29531.144} C_VEL
LIN {X 0,Y 116.212,Z 419.97,A -85,B 0,C 180,E1 -29532.148,E2 -29532.148} C_VEL
LIN {X 0,Y 113.258,Z 434.02,A -85,B 0,C 180,E1 -29532.74,E2 -29532.74} C_VEL
LIN {X 0,Y 109.332,Z 446.99,A -85,B 0,C 180,E1 -29533.531,E2 -29533.531} C_VEL
LIN {X 0,Y 104.422,Z 459.464,A -85,B 0,C 180,E1 -29534.653,E2 -29534.653} C_VEL
LIN {X 0,Y 97.934,Z 472.507,A -85,B 0,C 180,E1 -29536.298,E2 -29536.298} C_VEL
LIN {X 0,Y 91.776,Z 482.971,A -85,B 0,C 180,E1 -29538.296,E2 -29538.296} C_VEL
LIN {X 0,Y 84.548,Z 493.197,A -85,B 0,C 180,E1 -29540.75,E2 -29540.75} C_VEL
LIN {X 0,Y 76.98,Z 502.581,A -85,B 0,C 180,E1 -29544.084,E2 -29544.084} C_VEL
LIN {X 0,Y 68.301,Z 511.949,A -85,B 0,C 180,E1 -29549.001,E2 -29549.001} C_VEL
LIN {X 0,Y 60.293,Z 519.742,A -85,B 0,C 180,E1 -29555.32,E2 -29555.32} C_VEL
LIN {X 0,Y 53.207,Z 526.213,A -85,B 0,C 180,E1 -29563.408,E2 -29563.408} C_VEL
LIN {X 0,Y 47.391,Z 531.511,A -85,B 0,C 180,E1 -29573.616,E2 -29573.616} C_VEL
LIN {X 0,Y 42.486,Z 537.076,A -85,B 0,C 180,E1 -29590.679,E2 -29590.679} C_VEL
LIN {X 0,Y 41.439,Z 539.23,A -85,B 0,C 180,E1 -29600.235,E2 -29600.235} C_VEL
LIN {X 0,Y 41.34,Z 540.988,A -85,B 0,C 180,E1 -29609.999,E2 -29609.999} C_VEL
LIN {X 0,Y 41.512,Z 542.347,A -85,B 0,C 180,E1 -29619.746,E2 -29619.746} C_VEL
LIN {X 0,Y 44.654,Z 544.044,A -85,B 0,C 180,E1 -29638.173,E2 -29638.173} C_VEL
LIN {X 0,Y 51.504,Z 544.451,A -85,B 0,C 180,E1 -29653.019,E2 -29653.019} C_VEL
LIN {X 0,Y 60.941,Z 543.583,A -85,B 0,C 180,E1 -29663.827,E2 -29663.827} C_VEL
LIN {X 0,Y 71.927,Z 541.424,A -85,B 0,C 180,E1 -29671.566,E2 -29671.566} C_VEL
LIN {X 0,Y 83.915,Z 537.92,A -85,B 0,C 180,E1 -29677.107,E2 -29677.107} C_VEL
LIN {X 0,Y 96.497,Z 532.968,A -85,B 0,C 180,E1 -29681.222,E2 -29681.222} C_VEL
LIN {X 0,Y 109.56,Z 526.416,A -85,B 0,C 180,E1 -29684.192,E2 -29684.192} C_VEL
LIN {X 0,Y 121.154,Z 519.17,A -85,B 0,C 180,E1 -29686.317,E2 -29686.317} C_VEL
LIN {X 0,Y 132.871,Z 510.25,A -85,B 0,C 180,E1 -29688.097,E2 -29688.097} C_VEL
LIN {X 0,Y 143.062,Z 500.908,A -85,B 0,C 180,E1 -29689.259,E2 -29689.259} C_VEL
LIN {X 0,Y 153.309,Z 489.54,A -85,B 0,C 180,E1 -29690.257,E2 -29690.257} C_VEL
LIN {X 0,Y 161.861,Z 478.013,A -85,B 0,C 180,E1 -29691.033,E2 -29691.033} C_VEL
LIN {X 0,Y 169.625,Z 465.197,A -85,B 0,C 180,E1 -29691.561,E2 -29691.561} C_VEL
LIN {X 0,Y 175.662,Z 452.696,A -85,B 0,C 180,E1 -29691.966,E2 -29691.966} C_VEL
LIN {X 0,Y 179.375,Z 443.167,A -85,B 0,C 180,E1 -29692.213,E2 -29692.213} C_VEL
LIN {X 0,Y 179.776,Z 441.922,A -85,B 0,C 180,E1 -29692.474,E2 -29692.474} C_VEL
LIN {X 0,Y 179.771,Z 441.861,A -85,B 0,C 180,E1 -29694.149,E2 -29694.149} C_VEL
LIN {X 0,Y 174.702,Z 454.723,A -85,B 0,C 180,E1 -29694.642,E2 -29694.642} C_VEL
LIN {X 0,Y 168.33,Z 467.345,A -85,B 0,C 180,E1 -29695.207,E2 -29695.207} C_VEL
LIN {X 0,Y 162.974,Z 476.113,A -85,B 0,C 180,E1 -29695.717,E2 -29695.717} C_VEL
LIN {X 0,Y 159.583,Z 481.04,A -85,B 0,C 180,E1 -29695.807,E2 -29695.807} C_VEL
LIN {X 0,Y 153.51,Z 488.825,A -85,B 0,C 180,E1 -29695.324,E2 -29695.324} C_VEL
LIN {X 0,Y 147.076,Z 496.154,A -85,B 0,C 180,E1 -29694.844,E2 -29694.844} C_VEL
LIN {X 0,Y 142.991,Z 500.32,A -85,B 0,C 180,E1 -29694.982,E2 -29694.982} C_VEL
LIN {X 0,Y 132.073,Z 510.108,A -85,B 0,C 180,E1 -29696.128,E2 -29696.128} C_VEL
LIN {X 0,Y 121.345,Z 518.064,A -85,B 0,C 180,E1 -29697.503,E2 -29697.503} C_VEL
LIN {X 0,Y 110.522,Z 524.73,A -85,B 0,C 180,E1 -29699.216,E2 -29699.216} C_VEL
LIN {X 0,Y 98.427,Z 530.805,A -85,B 0,C 180,E1 -29701.589,E2 -29701.589} C_VEL
LIN {X 0,Y 86.476,Z 535.537,A -85,B 0,C 180,E1 -29704.655,E2 -29704.655} C_VEL
LIN {X 0,Y 77.972,Z 538.158,A -85,B 0,C 180,E1 -29707.497,E2 -29707.497} C_VEL
LIN {X 0,Y 65.038,Z 541.085,A -85,B 0,C 180,E1 -29713.466,E2 -29713.466} C_VEL
LIN {X 0,Y 53.113,Z 542.548,A -85,B 0,C 180,E1 -29722.149,E2 -29722.149} C_VEL
LIN {X 0,Y 42.971,Z 542.592,A -85,B 0,C 180,E1 -29735.143,E2 -29735.143} C_VEL
LIN {X 0,Y 35.987,Z 541.213,A -85,B 0,C 180,E1 -29754.138,E2 -29754.138} C_VEL
LIN {X 0,Y 33.6,Z 538.406,A -85,B 0,C 180,E1 -29777.928,E2 -29777.928} C_VEL
LIN {X 0,Y 35.245,Z 535.568,A -85,B 0,C 180,E1 -29794.631,E2 -29794.631} C_VEL
LIN {X 0,Y 39.461,Z 531.448,A -85,B 0,C 180,E1 -29810.868,E2 -29810.868} C_VEL
LIN {X 0,Y 45.382,Z 526.635,A -85,B 0,C 180,E1 -29822.822,E2 -29822.822} C_VEL
LIN {X 0,Y 54.017,Z 519.673,A -85,B 0,C 180,E1 -29833.083,E2 -29833.083} C_VEL
LIN {X 0,Y 62.364,Z 512.402,A -85,B 0,C 180,E1 -29839.524,E2 -29839.524} C_VEL
LIN {X 0,Y 71.265,Z 503.653,A -85,B 0,C 180,E1 -29844.449,E2 -29844.449} C_VEL
LIN {X 0,Y 79.539,Z 494.299,A -85,B 0,C 180,E1 -29847.928,E2 -29847.928} C_VEL
LIN {X 0,Y 85.309,Z 486.819,A -85,B 0,C 180,E1 -29849.955,E2 -29849.955} C_VEL
LIN {X 0,Y 93.197,Z 474.902,A -85,B 0,C 180,E1 -29852.382,E2 -29852.382} C_VEL
LIN {X 0,Y 99.58,Z 463.142,A -85,B 0,C 180,E1 -29854.136,E2 -29854.136} C_VEL
LIN {X 0,Y 105.442,Z 450.136,A -85,B 0,C 180,E1 -29855.248,E2 -29855.248} C_VEL
LIN {X 0,Y 110.143,Z 435.994,A -85,B 0,C 180,E1 -29856.316,E2 -29856.316} C_VEL
LIN {X 0,Y 113.5,Z 421.779,A -85,B 0,C 180,E1 -29856.98,E2 -29856.98} C_VEL
LIN {X 0,Y 116.135,Z 402.899,A -85,B 0,C 180,E1 -29857.495,E2 -29857.495} C_VEL
LIN {X 0,Y 117.406,Z 391.542,A -85,B 0,C 180,E1 -29857.857,E2 -29857.857} C_VEL
LIN {X 0,Y 116.225,Z 387.442,A -85,B 0,C 180,E1 -29861.496,E2 -29861.496} C_VEL
LIN {X 0,Y 115.391,Z 384.885,A -85,B 0,C 180,E1 -29864.956,E2 -29864.956} C_VEL
LIN {X 0,Y 114.841,Z 382.458,A -85,B 0,C 180,E1 -29869.426,E2 -29869.426} C_VEL
LIN {X 0,Y 114.695,Z 382.112,A -85,B 0,C 180,E1 -29872.965,E2 -29872.965} C_VEL
LIN {X 0,Y 114.956,Z 382.316,A -85,B 0,C 180,E1 -29876.997,E2 -29876.997} C_VEL
LIN {X 0,Y 115.67,Z 385.503,A -85,B 0,C 180,E1 -29881.887,E2 -29881.887} C_VEL
LIN {X 0,Y 116.814,Z 389.425,A -85,B 0,C 180,E1 -29886.057,E2 -29886.057} C_VEL
LIN {X 0,Y 117.508,Z 391.798,A -85,B 0,C 180,E1 -29888.009,E2 -29888.009} C_VEL
LIN {X 0,Y 113.999,Z 420.351,A -85,B 0,C 180,E1 -29888.796,E2 -29888.796} C_VEL
LIN {X 0,Y 110.967,Z 434.255,A -85,B 0,C 180,E1 -29889.311,E2 -29889.311} C_VEL
LIN {X 0,Y 107.038,Z 446.891,A -85,B 0,C 180,E1 -29889.98,E2 -29889.98} C_VEL
LIN {X 0,Y 102.007,Z 459.345,A -85,B 0,C 180,E1 -29890.955,E2 -29890.955} C_VEL
LIN {X 0,Y 95.34,Z 472.373,A -85,B 0,C 180,E1 -29892.389,E2 -29892.389} C_VEL
LIN {X 0,Y 88.274,Z 483.852,A -85,B 0,C 180,E1 -29894.385,E2 -29894.385} C_VEL
LIN {X 0,Y 81.475,Z 493.042,A -85,B 0,C 180,E1 -29896.337,E2 -29896.337} C_VEL
LIN {X 0,Y 72.772,Z 503.244,A -85,B 0,C 180,E1 -29899.678,E2 -29899.678} C_VEL
LIN {X 0,Y 63.633,Z 512.469,A -85,B 0,C 180,E1 -29904.333,E2 -29904.333} C_VEL
LIN {X 0,Y 54.164,Z 520.875,A -85,B 0,C 180,E1 -29911.278,E2 -29911.278} C_VEL
LIN {X 0,Y 46.162,Z 527.434,A -85,B 0,C 180,E1 -29920.427,E2 -29920.427} C_VEL
LIN {X 0,Y 39.956,Z 532.512,A -85,B 0,C 180,E1 -29932.003,E2 -29932.003} C_VEL
LIN {X 0,Y 34.999,Z 537.715,A -85,B 0,C 180,E1 -29952.469,E2 -29952.469} C_VEL
LIN {X 0,Y 34.252,Z 540.604,A -85,B 0,C 180,E1 -29969.999,E2 -29969.999} C_VEL
LIN {X 0,Y 34.516,Z 542.008,A -85,B 0,C 180,E1 -29981.747,E2 -29981.747} C_VEL
LIN {X 0,Y 38.519,Z 543.785,A -85,B 0,C 180,E1 -30003.184,E2 -30003.184} C_VEL
LIN {X 0,Y 46.541,Z 544.27,A -85,B 0,C 180,E1 -30019.025,E2 -30019.025} C_VEL
LIN {X 0,Y 57.019,Z 543.479,A -85,B 0,C 180,E1 -30029.628,E2 -30029.628} C_VEL
LIN {X 0,Y 68.811,Z 541.398,A -85,B 0,C 180,E1 -30036.806,E2 -30036.806} C_VEL
LIN {X 0,Y 81.404,Z 537.976,A -85,B 0,C 180,E1 -30041.741,E2 -30041.741} C_VEL
LIN {X 0,Y 94.45,Z 533.11,A -85,B 0,C 180,E1 -30045.306,E2 -30045.306} C_VEL
LIN {X 0,Y 107.841,Z 526.65,A -85,B 0,C 180,E1 -30047.829,E2 -30047.829} C_VEL
LIN {X 0,Y 119.678,Z 519.503,A -85,B 0,C 180,E1 -30049.61,E2 -30049.61} C_VEL
LIN {X 0,Y 131.596,Z 510.716,A -85,B 0,C 180,E1 -30051.107,E2 -30051.107} C_VEL
LIN {X 0,Y 141.917,Z 501.524,A -85,B 0,C 180,E1 -30052.058,E2 -30052.058} C_VEL
LIN {X 0,Y 151.412,Z 491.396,A -85,B 0,C 180,E1 -30052.803,E2 -30052.803} C_VEL
LIN {X 0,Y 155.722,Z 486.123,A -85,B 0,C 180,E1 -30053.152,E2 -30053.152} C_VEL
LIN {X 0,Y 155.524,Z 486.333,A -85,B 0,C 180,E1 -30053.79,E2 -30053.79} C_VEL
LIN {X 0,Y 146.474,Z 496.771,A -85,B 0,C 180,E1 -30054.64,E2 -30054.64} C_VEL
LIN {X 0,Y 142.991,Z 500.32,A -85,B 0,C 180,E1 -30054.982,E2 -30054.982} C_VEL
LIN {X 0,Y 138.16,Z 504.951,A -85,B 0,C 180,E1 -30055.202,E2 -30055.202} C_VEL
LIN {X 0,Y 129.522,Z 512.117,A -85,B 0,C 180,E1 -30054.84,E2 -30054.84} C_VEL
LIN {X 0,Y 120.389,Z 518.634,A -85,B 0,C 180,E1 -30054.499,E2 -30054.499} C_VEL
LIN {X 0,Y 114.769,Z 522.165,A -85,B 0,C 180,E1 -30054.863,E2 -30054.863} C_VEL
LIN {X 0,Y 101.85,Z 529.046,A -85,B 0,C 180,E1 -30056.684,E2 -30056.684} C_VEL
LIN {X 0,Y 91.389,Z 533.551,A -85,B 0,C 180,E1 -30058.58,E2 -30058.58} C_VEL
LIN {X 0,Y 80.832,Z 537.131,A -85,B 0,C 180,E1 -30061.012,E2 -30061.012} C_VEL
LIN {X 0,Y 65.419,Z 540.859,A -85,B 0,C 180,E1 -30066.159,E2 -30066.159} C_VEL
LIN {X 0,Y 57.121,Z 542.1,A -85,B 0,C 180,E1 -30070.178,E2 -30070.178} C_VEL
LIN {X 0,Y 44.74,Z 542.935,A -85,B 0,C 180,E1 -30079.53,E2 -30079.53} C_VEL
LIN {X 0,Y 34.243,Z 542.358,A -85,B 0,C 180,E1 -30094.823,E2 -30094.823} C_VEL
LIN {X 0,Y 30.312,Z 541.541,A -85,B 0,C 180,E1 -30105.932,E2 -30105.932} C_VEL
LIN {X 0,Y 27.593,Z 540.375,A -85,B 0,C 180,E1 -30119.379,E2 -30119.379} C_VEL
LIN {X 0,Y 27.219,Z 536.937,A -85,B 0,C 180,E1 -30150.002,E2 -30150.002} C_VEL
LIN {X 0,Y 31.083,Z 533.395,A -85,B 0,C 180,E1 -30169.827,E2 -30169.827} C_VEL
LIN {X 0,Y 37.171,Z 528.955,A -85,B 0,C 180,E1 -30184.557,E2 -30184.557} C_VEL
LIN {X 0,Y 46.217,Z 522.532,A -85,B 0,C 180,E1 -30196.246,E2 -30196.246} C_VEL
LIN {X 0,Y 56.471,Z 514.548,A -85,B 0,C 180,E1 -30203.993,E2 -30203.993} C_VEL
LIN {X 0,Y 65.798,Z 506.194,A -85,B 0,C 180,E1 -30208.703,E2 -30208.703} C_VEL
LIN {X 0,Y 75.755,Z 495.77,A -85,B 0,C 180,E1 -30212.372,E2 -30212.372} C_VEL
LIN {X 0,Y 82.43,Z 487.501,A -85,B 0,C 180,E1 -30214.401,E2 -30214.401} C_VEL
LIN {X 0,Y 90.134,Z 476.4,A -85,B 0,C 180,E1 -30216.373,E2 -30216.373} C_VEL
LIN {X 0,Y 96.695,Z 464.935,A -85,B 0,C 180,E1 -30217.924,E2 -30217.924} C_VEL
LIN {X 0,Y 101.821,Z 454.337,A -85,B 0,C 180,E1 -30218.717,E2 -30218.717} C_VEL
LIN {X 0,Y 106.712,Z 441.43,A -85,B 0,C 180,E1 -30219.604,E2 -30219.604} C_VEL
LIN {X 0,Y 110.685,Z 427.112,A -85,B 0,C 180,E1 -30220.301,E2 -30220.301} C_VEL
LIN {X 0,Y 113.208,Z 413.244,A -85,B 0,C 180,E1 -30220.708,E2 -30220.708} C_VEL
LIN {X 0,Y 115.324,Z 395.532,A -85,B 0,C 180,E1 -30221.177,E2 -30221.177} C_VEL
LIN {X 0,Y 114.443,Z 392.095,A -85,B 0,C 180,E1 -30225.104,E2 -30225.104} C_VEL
LIN {X 0,Y 113.895,Z 389.435,A -85,B 0,C 180,E1 -30230.171,E2 -30230.171} C_VEL
LIN {X 0,Y 113.848,Z 389.181,A -85,B 0,C 180,E1 -30234.329,E2 -30234.329} C_VEL
LIN {X 0,Y 114.019,Z 389.511,A -85,B 0,C 180,E1 -30236.721,E2 -30236.721} C_VEL
LIN {X 0,Y 114.547,Z 392.342,A -85,B 0,C 180,E1 -30241.018,E2 -30241.018} C_VEL
LIN {X 0,Y 115.394,Z 395.846,A -85,B 0,C 180,E1 -30244.711,E2 -30244.711} C_VEL
LIN {X 0,Y 112.204,Z 420.667,A -85,B 0,C 180,E1 -30245.327,E2 -30245.327} C_VEL
LIN {X 0,Y 108.841,Z 435.379,A -85,B 0,C 180,E1 -30245.789,E2 -30245.789} C_VEL
LIN {X 0,Y 104.74,Z 447.922,A -85,B 0,C 180,E1 -30246.332,E2 -30246.332} C_VEL
LIN {X 0,Y 99.182,Z 461.015,A -85,B 0,C 180,E1 -30247.242,E2 -30247.242} C_VEL
LIN {X 0,Y 92.359,Z 473.676,A -85,B 0,C 180,E1 -30248.422,E2 -30248.422} C_VEL
LIN {X 0,Y 84.814,Z 485.299,A -85,B 0,C 180,E1 -30250.263,E2 -30250.263} C_VEL
LIN {X 0,Y 78.916,Z 492.882,A -85,B 0,C 180,E1 -30251.591,E2 -30251.591} C_VEL
LIN {X 0,Y 70.684,Z 502.257,A -85,B 0,C 180,E1 -30254.207,E2 -30254.207} C_VEL
LIN {X 0,Y 61.027,Z 511.611,A -85,B 0,C 180,E1 -30258.18,E2 -30258.18} C_VEL
LIN {X 0,Y 51.677,Z 519.485,A -85,B 0,C 180,E1 -30263.753,E2 -30263.753} C_VEL
LIN {X 0,Y 44.57,Z 524.833,A -85,B 0,C 180,E1 -30269.859,E2 -30269.859} C_VEL
LIN {X 0,Y 36.87,Z 530.33,A -85,B 0,C 180,E1 -30280.317,E2 -30280.317} C_VEL
LIN {X 0,Y 29.382,Z 536.077,A -85,B 0,C 180,E1 -30301.419,E2 -30301.419} C_VEL
LIN {X 0,Y 27.524,Z 538.332,A -85,B 0,C 180,E1 -30315.205,E2 -30315.205} C_VEL
LIN {X 0,Y 27.138,Z 540.193,A -85,B 0,C 180,E1 -30329.998,E2 -30329.998} C_VEL
LIN {X 0,Y 27.597,Z 541.643,A -85,B 0,C 180,E1 -30344.752,E2 -30344.752} C_VEL
LIN {X 0,Y 32.777,Z 543.508,A -85,B 0,C 180,E1 -30370.032,E2 -30370.032} C_VEL
LIN {X 0,Y 42.209,Z 544.076,A -85,B 0,C 180,E1 -30386.354,E2 -30386.354} C_VEL
LIN {X 0,Y 53.756,Z 543.367,A -85,B 0,C 180,E1 -30396.224,E2 -30396.224} C_VEL
LIN {X 0,Y 66.329,Z 541.371,A -85,B 0,C 180,E1 -30402.472,E2 -30402.472} C_VEL
LIN {X 0,Y 79.46,Z 538.032,A -85,B 0,C 180,E1 -30406.628,E2 -30406.628} C_VEL
LIN {X 0,Y 92.903,Z 533.252,A -85,B 0,C 180,E1 -30409.545,E2 -30409.545} C_VEL
LIN {X 0,Y 106.569,Z 526.884,A -85,B 0,C 180,E1 -30411.567,E2 -30411.567} C_VEL
LIN {X 0,Y 118.606,Z 519.837,A -85,B 0,C 180,E1 -30412.973,E2 -30412.973} C_VEL
LIN {X 0,Y 123.189,Z 516.753,A -85,B 0,C 180,E1 -30413.444,E2 -30413.444} C_VEL
LIN {X 0,Y 122.086,Z 517.504,A -85,B 0,C 180,E1 -30414.004,E2 -30414.004} C_VEL
LIN {X 0,Y 114.769,Z 522.165,A -85,B 0,C 180,E1 -30414.863,E2 -30414.863} C_VEL
LIN {X 0,Y 108.529,Z 525.733,A -85,B 0,C 180,E1 -30415.361,E2 -30415.361} C_VEL
LIN {X 0,Y 97.593,Z 531.015,A -85,B 0,C 180,E1 -30415.293,E2 -30415.293} C_VEL
LIN {X 0,Y 88.563,Z 534.58,A -85,B 0,C 180,E1 -30415.175,E2 -30415.175} C_VEL
LIN {X 0,Y 81.729,Z 536.851,A -85,B 0,C 180,E1 -30415.653,E2 -30415.653} C_VEL
LIN {X 0,Y 79.478,Z 537.504,A -85,B 0,C 180,E1 -30416.026,E2 -30416.026} C_VEL
LIN {X 0,Y 70.316,Z 539.843,A -85,B 0,C 180,E1 -30418.108,E2 -30418.108} C_VEL
LIN {X 0,Y 56.282,Z 542.204,A -85,B 0,C 180,E1 -30422.651,E2 -30422.651} C_VEL
LIN {X 0,Y 42.822,Z 543.124,A -85,B 0,C 180,E1 -30430.038,E2 -30430.038} C_VEL
LIN {X 0,Y 30.6,Z 542.631,A -85,B 0,C 180,E1 -30443.27,E2 -30443.27} C_VEL
LIN {X 0,Y 25.511,Z 541.855,A -85,B 0,C 180,E1 -30454.267,E2 -30454.267} C_VEL
LIN {X 0,Y 19.535,Z 539.259,A -85,B 0,C 180,E1 -30488.917,E2 -30488.917} C_VEL
LIN {X 0,Y 21.657,Z 535.854,A -85,B 0,C 180,E1 -30523.323,E2 -30523.323} C_VEL
LIN {X 0,Y 28.994,Z 531.127,A -85,B 0,C 180,E1 -30547.302,E2 -30547.302} C_VEL
LIN {X 0,Y 37.11,Z 526.13,A -85,B 0,C 180,E1 -30559.247,E2 -30559.247} C_VEL
LIN {X 0,Y 47.81,Z 518.955,A -85,B 0,C 180,E1 -30567.697,E2 -30567.697} C_VEL
LIN {X 0,Y 57.475,Z 511.444,A -85,B 0,C 180,E1 -30572.439,E2 -30572.439} C_VEL
LIN {X 0,Y 67.382,Z 502.421,A -85,B 0,C 180,E1 -30575.87,E2 -30575.87} C_VEL
LIN {X 0,Y 76.715,Z 492.307,A -85,B 0,C 180,E1 -30578.397,E2 -30578.397} C_VEL
LIN {X 0,Y 85.018,Z 481.599,A -85,B 0,C 180,E1 -30580.103,E2 -30580.103} C_VEL
LIN {X 0,Y 92.557,Z 469.759,A -85,B 0,C 180,E1 -30581.647,E2 -30581.647} C_VEL
LIN {X 0,Y 99.421,Z 456.564,A -85,B 0,C 180,E1 -30582.611,E2 -30582.611} C_VEL
LIN {X 0,Y 102.904,Z 448.344,A -85,B 0,C 180,E1 -30582.968,E2 -30582.968} C_VEL
LIN {X 0,Y 107.712,Z 433.791,A -85,B 0,C 180,E1 -30583.716,E2 -30583.716} C_VEL
LIN {X 0,Y 110.852,Z 420.165,A -85,B 0,C 180,E1 -30584.127,E2 -30584.127} C_VEL
LIN {X 0,Y 113.583,Z 400.038,A -85,B 0,C 180,E1 -30584.587,E2 -30584.587} C_VEL
LIN {X 0,Y 113.123,Z 397.858,A -85,B 0,C 180,E1 -30587.902,E2 -30587.902} C_VEL
LIN {X 0,Y 112.972,Z 396.392,A -85,B 0,C 180,E1 -30590.929,E2 -30590.929} C_VEL
LIN {X 0,Y 113.064,Z 396.392,A -85,B 0,C 180,E1 -30595.903,E2 -30595.903} C_VEL
LIN {X 0,Y 113.431,Z 399.089,A -85,B 0,C 180,E1 -30600.005,E2 -30600.005} C_VEL
LIN {X 0,Y 113.636,Z 400.205,A -85,B 0,C 180,E1 -30601.302,E2 -30601.302} C_VEL
LIN {X 0,Y 110.781,Z 421.263,A -85,B 0,C 180,E1 -30601.77,E2 -30601.77} C_VEL
LIN {X 0,Y 107.342,Z 435.811,A -85,B 0,C 180,E1 -30602.126,E2 -30602.126} C_VEL
LIN {X 0,Y 103.321,Z 447.823,A -85,B 0,C 180,E1 -30602.508,E2 -30602.508} C_VEL
LIN {X 0,Y 97.666,Z 460.896,A -85,B 0,C 180,E1 -30603.214,E2 -30603.214} C_VEL
LIN {X 0,Y 90.938,Z 473.179,A -85,B 0,C 180,E1 -30604.087,E2 -30604.087} C_VEL
LIN {X 0,Y 83.83,Z 483.956,A -85,B 0,C 180,E1 -30605.414,E2 -30605.414} C_VEL
LIN {X 0,Y 76.936,Z 492.727,A -85,B 0,C 180,E1 -30606.583,E2 -30606.583} C_VEL
LIN {X 0,Y 67.576,Z 502.92,A -85,B 0,C 180,E1 -30608.886,E2 -30608.886} C_VEL
LIN {X 0,Y 57.52,Z 512.131,A -85,B 0,C 180,E1 -30612.19,E2 -30612.19} C_VEL
LIN {X 0,Y 46.69,Z 520.537,A -85,B 0,C 180,E1 -30617.533,E2 -30617.533} C_VEL
LIN {X 0,Y 38.434,Z 526.153,A -85,B 0,C 180,E1 -30623.893,E2 -30623.893} C_VEL
LIN {X 0,Y 30.002,Z 531.376,A -85,B 0,C 180,E1 -30634.927,E2 -30634.927} C_VEL
LIN {X 0,Y 23.353,Z 535.576,A -85,B 0,C 180,E1 -30652.993,E2 -30652.993} C_VEL
LIN {X 0,Y 20.703,Z 537.875,A -85,B 0,C 180,E1 -30670.153,E2 -30670.153} C_VEL
LIN {X 0,Y 20.028,Z 539.779,A -85,B 0,C 180,E1 -30689.998,E2 -30689.998} C_VEL
LIN {X 0,Y 20.815,Z 541.27,A -85,B 0,C 180,E1 -30709.73,E2 -30709.73} C_VEL
LIN {X 0,Y 27.698,Z 543.211,A -85,B 0,C 180,E1 -30739.566,E2 -30739.566} C_VEL
LIN {X 0,Y 38.717,Z 543.858,A -85,B 0,C 180,E1 -30755.17,E2 -30755.17} C_VEL
LIN {X 0,Y 51.293,Z 543.229,A -85,B 0,C 180,E1 -30763.551,E2 -30763.551} C_VEL
LIN {X 0,Y 64.541,Z 541.319,A -85,B 0,C 180,E1 -30768.52,E2 -30768.52} C_VEL
LIN {X 0,Y 78.121,Z 538.08,A -85,B 0,C 180,E1 -30771.713,E2 -30771.713} C_VEL
LIN {X 0,Y 84.98,Z 535.927,A -85,B 0,C 180,E1 -30772.928,E2 -30772.928} C_VEL
LIN {X 0,Y 89.32,Z 534.333,A -85,B 0,C 180,E1 -30774.303,E2 -30774.303} C_VEL
LIN {X 0,Y 79.478,Z 537.504,A -85,B 0,C 180,E1 -30776.026,E2 -30776.026} C_VEL
LIN {X 0,Y 73.518,Z 539.127,A -85,B 0,C 180,E1 -30776.773,E2 -30776.773} C_VEL
LIN {X 0,Y 63.252,Z 541.264,A -85,B 0,C 180,E1 -30776.762,E2 -30776.762} C_VEL
LIN {X 0,Y 54.938,Z 542.446,A -85,B 0,C 180,E1 -30776.637,E2 -30776.637} C_VEL
LIN {X 0,Y 48.748,Z 543.018,A -85,B 0,C 180,E1 -30777.437,E2 -30777.437} C_VEL
LIN {X 0,Y 46.733,Z 543.102,A -85,B 0,C 180,E1 -30778.066,E2 -30778.066} C_VEL
LIN {X 0,Y 35.216,Z 543.285,A -85,B 0,C 180,E1 -30783.793,E2 -30783.793} C_VEL
LIN {X 0,Y 21.942,Z 542.133,A -85,B 0,C 180,E1 -30798.654,E2 -30798.654} C_VEL
LIN {X 0,Y 12.976,Z 539.653,A -85,B 0,C 180,E1 -30837.211,E2 -30837.211} C_VEL
LIN {X 0,Y 15.298,Z 535.998,A -85,B 0,C 180,E1 -30893.339,E2 -30893.339} C_VEL
LIN {X 0,Y 23.701,Z 531.69,A -85,B 0,C 180,E1 -30917.846,E2 -30917.846} C_VEL
LIN {X 0,Y 32.905,Z 526.788,A -85,B 0,C 180,E1 -30928.688,E2 -30928.688} C_VEL
LIN {X 0,Y 44.427,Z 519.716,A -85,B 0,C 180,E1 -30935.451,E2 -30935.451} C_VEL
LIN {X 0,Y 56.252,Z 510.965,A -85,B 0,C 180,E1 -30939.557,E2 -30939.557} C_VEL
LIN {X 0,Y 66.52,Z 501.806,A -85,B 0,C 180,E1 -30941.963,E2 -30941.963} C_VEL
LIN {X 0,Y 75.375,Z 492.375,A -85,B 0,C 180,E1 -30943.651,E2 -30943.651} C_VEL
LIN {X 0,Y 83.736,Z 481.805,A -85,B 0,C 180,E1 -30944.837,E2 -30944.837} C_VEL
LIN {X 0,Y 91.441,Z 469.966,A -85,B 0,C 180,E1 -30946.007,E2 -30946.007} C_VEL
LIN {X 0,Y 98.402,Z 456.777,A -85,B 0,C 180,E1 -30946.681,E2 -30946.681} C_VEL
LIN {X 0,Y 102.286,Z 447.611,A -85,B 0,C 180,E1 -30946.942,E2 -30946.942} C_VEL
LIN {X 0,Y 107.074,Z 433.092,A -85,B 0,C 180,E1 -30947.503,E2 -30947.503} C_VEL
LIN {X 0,Y 110.212,Z 419.285,A -85,B 0,C 180,E1 -30947.788,E2 -30947.788} C_VEL
LIN {X 0,Y 112.195,Z 405.036,A -85,B 0,C 180,E1 -30948.087,E2 -30948.087} C_VEL
LIN {X 0,Y 112.083,Z 403.477,A -85,B 0,C 180,E1 -30950.986,E2 -30950.986} C_VEL
LIN {X 0,Y 112.094,Z 403.264,A -85,B 0,C 180,E1 -30954.404,E2 -30954.404} C_VEL
LIN {X 0,Y 112.163,Z 404.045,A -85,B 0,C 180,E1 -30956.412,E2 -30956.412} C_VEL
LIN {X 0,Y 112.254,Z 404.888,A -85,B 0,C 180,E1 -30957.807,E2 -30957.807} C_VEL
LIN {X 0,Y 109.602,Z 422.85,A -85,B 0,C 180,E1 -30958.133,E2 -30958.133} C_VEL
LIN {X 0,Y 106.068,Z 437.012,A -85,B 0,C 180,E1 -30958.375,E2 -30958.375} C_VEL
LIN {X 0,Y 101.935,Z 448.855,A -85,B 0,C 180,E1 -30958.609,E2 -30958.609} C_VEL
LIN {X 0,Y 96.646,Z 460.776,A -85,B 0,C 180,E1 -30959.079,E2 -30959.079} C_VEL
LIN {X 0,Y 89.805,Z 473.088,A -85,B 0,C 180,E1 -30959.656,E2 -30959.656} C_VEL
LIN {X 0,Y 82.583,Z 483.808,A -85,B 0,C 180,E1 -30960.603,E2 -30960.603} C_VEL
LIN {X 0,Y 75.571,Z 492.571,A -85,B 0,C 180,E1 -30961.353,E2 -30961.353} C_VEL
LIN {X 0,Y 66.847,Z 501.934,A -85,B 0,C 180,E1 -30962.824,E2 -30962.824} C_VEL
LIN {X 0,Y 56.442,Z 511.273,A -85,B 0,C 180,E1 -30965.046,E2 -30965.046} C_VEL
LIN {X 0,Y 46.17,Z 519.049,A -85,B 0,C 180,E1 -30968.374,E2 -30968.374} C_VEL
LIN {X 0,Y 36.129,Z 525.502,A -85,B 0,C 180,E1 -30973.438,E2 -30973.438} C_VEL
LIN {X 0,Y 26.558,Z 530.785,A -85,B 0,C 180,E1 -30982.148,E2 -30982.148} C_VEL
LIN {X 0,Y 15.94,Z 536.331,A -85,B 0,C 180,E1 -31008.593,E2 -31008.593} C_VEL
LIN {X 0,Y 12.931,Z 539.365,A -85,B 0,C 180,E1 -31049.996,E2 -31049.996} C_VEL
LIN {X 0,Y 14.319,Z 540.895,A -85,B 0,C 180,E1 -31079.389,E2 -31079.389} C_VEL
LIN {X 0,Y 23.695,Z 542.913,A -85,B 0,C 180,E1 -31112.841,E2 -31112.841} C_VEL
LIN {X 0,Y 36.306,Z 543.638,A -85,B 0,C 180,E1 -31125.428,E2 -31125.428} C_VEL
LIN {X 0,Y 49.744,Z 543.086,A -85,B 0,C 180,E1 -31131.47,E2 -31131.47} C_VEL
LIN {X 0,Y 56.598,Z 542.331,A -85,B 0,C 180,E1 -31133.39,E2 -31133.39} C_VEL
LIN {X 0,Y 56.435,Z 542.308,A -85,B 0,C 180,E1 -31135.019,E2 -31135.019} C_VEL
LIN {X 0,Y 46.733,Z 543.102,A -85,B 0,C 180,E1 -31138.066,E2 -31138.066} C_VEL
LIN {X 0,Y 40.945,Z 543.366,A -85,B 0,C 180,E1 -31139.578,E2 -31139.578} C_VEL
LIN {X 0,Y 31.036,Z 543.262,A -85,B 0,C 180,E1 -31139.991,E2 -31139.991} C_VEL
LIN {X 0,Y 23.086,Z 542.683,A -85,B 0,C 180,E1 -31140.042,E2 -31140.042} C_VEL
LIN {X 0,Y 17.254,Z 541.981,A -85,B 0,C 180,E1 -31142.479,E2 -31142.479} C_VEL
LIN {X 0,Y 15.389,Z 541.642,A -85,B 0,C 180,E1 -31144.598,E2 -31144.598} C_VEL
LIN {X 0,Y 7.877,Z 540.049,A -85,B 0,C 180,E1 -31166.862,E2 -31166.862} C_VEL
LIN {X 0,Y 10.038,Z 536.128,A -85,B 0,C 180,E1 -31275.639,E2 -31275.639} C_VEL
LIN {X 0,Y 19.622,Z 532.254,A -85,B 0,C 180,E1 -31293.564,E2 -31293.564} C_VEL
LIN {X 0,Y 29.832,Z 527.445,A -85,B 0,C 180,E1 -31300.452,E2 -31300.452} C_VEL
LIN {X 0,Y 41.97,Z 520.481,A -85,B 0,C 180,E1 -31304.332,E2 -31304.332} C_VEL
LIN {X 0,Y 52.433,Z 513.211,A -85,B 0,C 180,E1 -31306.353,E2 -31306.353} C_VEL
LIN {X 0,Y 62.921,Z 504.464,A -85,B 0,C 180,E1 -31307.774,E2 -31307.774} C_VEL
LIN {X 0,Y 72.682,Z 494.691,A -85,B 0,C 180,E1 -31308.822,E2 -31308.822} C_VEL
LIN {X 0,Y 79.552,Z 486.624,A -85,B 0,C 180,E1 -31309.367,E2 -31309.367} C_VEL
LIN {X 0,Y 88.264,Z 474.42,A -85,B 0,C 180,E1 -31310.179,E2 -31310.179} C_VEL
LIN {X 0,Y 95.246,Z 462.323,A -85,B 0,C 180,E1 -31310.716,E2 -31310.716} C_VEL
LIN {X 0,Y 100.984,Z 449.919,A -85,B 0,C 180,E1 -31310.841,E2 -31310.841} C_VEL
LIN {X 0,Y 105.909,Z 435.86,A -85,B 0,C 180,E1 -31311.233,E2 -31311.233} C_VEL
LIN {X 0,Y 109.432,Z 421.472,A -85,B 0,C 180,E1 -31311.436,E2 -31311.436} C_VEL
LIN {X 0,Y 111.184,Z 410.438,A -85,B 0,C 180,E1 -31311.657,E2 -31311.657} C_VEL
LIN {X 0,Y 111.206,Z 410.306,A -85,B 0,C 180,E1 -31314.217,E2 -31314.217} C_VEL
LIN {X 0,Y 108.746,Z 425.047,A -85,B 0,C 180,E1 -31314.449,E2 -31314.449} C_VEL
LIN {X 0,Y 104.774,Z 439.632,A -85,B 0,C 180,E1 -31314.587,E2 -31314.587} C_VEL
LIN {X 0,Y 99.697,Z 453.031,A -85,B 0,C 180,E1 -31314.691,E2 -31314.691} C_VEL
LIN {X 0,Y 93.485,Z 465.705,A -85,B 0,C 180,E1 -31314.93,E2 -31314.93} C_VEL
LIN {X 0,Y 85.78,Z 478.26,A -85,B 0,C 180,E1 -31315.307,E2 -31315.307} C_VEL
LIN {X 0,Y 79.279,Z 487.115,A -85,B 0,C 180,E1 -31315.782,E2 -31315.782} C_VEL
LIN {X 0,Y 73.968,Z 493.412,A -85,B 0,C 180,E1 -31316.062,E2 -31316.062} C_VEL
LIN {X 0,Y 65.109,Z 502.596,A -85,B 0,C 180,E1 -31316.813,E2 -31316.813} C_VEL
LIN {X 0,Y 54.501,Z 511.794,A -85,B 0,C 180,E1 -31317.975,E2 -31317.975} C_VEL
LIN {X 0,Y 42.168,Z 520.57,A -85,B 0,C 180,E1 -31320.073,E2 -31320.073} C_VEL
LIN {X 0,Y 31.676,Z 526.717,A -85,B 0,C 180,E1 -31323.23,E2 -31323.23} C_VEL
LIN {X 0,Y 21.345,Z 531.776,A -85,B 0,C 180,E1 -31328.965,E2 -31328.965} C_VEL
LIN {X 0,Y 8.764,Z 536.964,A -85,B 0,C 180,E1 -31356.683,E2 -31356.683} C_VEL
LIN {X 0,Y 5.822,Z 538.952,A -85,B 0,C 180,E1 -31409.992,E2 -31409.992} C_VEL
LIN {X 0,Y 8.845,Z 540.522,A -85,B 0,C 180,E1 -31462.607,E2 -31462.607} C_VEL
LIN {X 0,Y 21.4,Z 542.616,A -85,B 0,C 180,E1 -31490.124,E2 -31490.124} C_VEL
LIN {X 0,Y 25.983,Z 543.007,A -85,B 0,C 180,E1 -31495.359,E2 -31495.359} C_VEL
LIN {X 0,Y 15.389,Z 541.642,A -85,B 0,C 180,E1 -31504.598,E2 -31504.598} C_VEL
LIN {X 0,Y 13.277,Z 543.62,A -85,B 0,C 180,E1 -31508.192,E2 -31508.192} C_VEL
LIN {X 0,Y 13.277,Z 600,A -85,B 0,C 180,E1 -31508.192,E2 -31508.192} C_VEL
LIN {X 0,Y 13.277,Z 600,A -85,B 0,C 180,E1 -31508.192,E2 -31508.192}

QRS_NEXT_CUT()

QRS_NEXT()
QRS_HOME()

END
